								IF arrAxisCtrl[AxiseNo.AxisName.TailCurlLine].Cmd.arrbRealPoint[1] THEN
									IF Mach_Control.WJ_b.SinStepMode THEN//尾卷单步模式
									TailCurlSinStep:=TRUE;
								ELSE
									TailCurlSinStep:=FALSE;
								END_IF	
									arrAxisCtrl[AxiseNo.AxisName.TailCurlLine].Cmd.iGoSetPos:=0;
									//Mach_Control.WJ_b.TailCultOffloadingDone:=TRUE;
									TailCurlStep3:=1305;
								ELSE
									arrAxisCtrl[AxiseNo.AxisName.TailCurlLine].Cmd.iGoSetPos:=1;//尾卷夹电芯平移至初始位
								END_IF
						END_IF	
				END_IF	

				1305:
							IF NOT TailCurlSinStep THEN			
								IF 	arrAxisCtrl[AxiseNo.AxisName.TailCurlUpDown].Status.Homed AND arrAxisCtrl[AxiseNo.AxisName.TailCurlUpDown].Status.NoMoving  THEN
									IF arrAxisCtrl[AxiseNo.AxisName.TailCurlUpDown].Cmd.arrbRealPoint[4] THEN
													arrAxisCtrl[AxiseNo.AxisName.TailCurlUpDown].Cmd.iGoSetPos:=0;
													IF Mach_Control.WJ_b.SinStepMode THEN//尾卷单步模式
													TailCurlSinStep:=TRUE;
													ELSE
														TailCurlSinStep:=FALSE;
													END_IF	
													TailCurlStep3:=1310;
									ELSE
													arrAxisCtrl[AxiseNo.AxisName.TailCurlUpDown].Cmd.iGoSetPos:=4;//尾卷夹电芯升降至下电芯位
									END_IF
								END_IF	
						END_IF	
				
				1310:
					IF NOT TailCurlSinStep THEN		
					 IF arrAxisCtrl[AxiseNo.AxisName.GluingLine].Status.fActPos<=arrAxispar[AxiseNo.AxisName.GluingLine].arrTargetPoint[10] 
						AND arrAxisCtrl[AxiseNo.AxisName.GluingLine].Status.Homed AND NOT Mach_Control.WJ_b.TailCultOffloading AND arrAxis[AxiseNo.AxisName.TailCurlWhirling].Status.Homed 
						AND arrAxisCtrl[AxiseNo.AxisName.TailCurlWhirling].Status.NoMoving AND arrAxisCtrl[AxiseNo.AxisName.TailCurlLine].Status.NoMoving AND arrAxisCtrl[AxiseNo.AxisName.TailCurlLine].Cmd.arrbRealPoint[1] THEN
						
								IF arrAxisCtrl[AxiseNo.AxisName.TailCurlWhirling].Cmd.arrbRealPoint[1] THEN
									IF Mach_Control.WJ_b.SinStepMode THEN//尾卷单步模式
									TailCurlSinStep:=TRUE;
								ELSE
									TailCurlSinStep:=FALSE;
								END_IF	
									arrAxisCtrl[AxiseNo.AxisName.TailCurlWhirling].Cmd.iGoSetPos:=0;
									
									TailCurlStep3:=1320;
								ELSE
									arrAxisCtrl[AxiseNo.AxisName.TailCurlWhirling].Cmd.iGoSetPos:=1;//尾卷夹电芯旋转至取电芯位
								END_IF
						END_IF	
				END_IF	
	
	            1320://尾卷夹电芯平移去取电芯等待位
					 IF NOT TailCurlSinStep THEN	
								 IF  arrAxisCtrl[AxiseNo.AxisName.TailCurlUpDown].Status.Homed AND arrAxisCtrl[AxiseNo.AxisName.TailCurlUpDown].Status.NoMoving THEN
												IF arrAxisCtrl[AxiseNo.AxisName.TailCurlUpDown].Cmd.arrbRealPoint[1] THEN
													arrAxisCtrl[AxiseNo.AxisName.TailCurlUpDown].Cmd.iGoSetPos:=0;
												ELSE
													arrAxisCtrl[AxiseNo.AxisName.TailCurlUpDown].Cmd.iGoSetPos:=1;//尾卷夹升降去取电芯高度
												END_IF
								 END_IF
							 
							   IF arrAxisCtrl[AxiseNo.AxisName.TailCurlWhirling].Cmd.arrbRealPoint[1] AND arrAxisCtrl[AxiseNo.AxisName.TailCurlUpDown].Cmd.arrbRealPoint[1] AND
								  arrAxisCtrl[AxiseNo.AxisName.TailCurlSEPTALine].Cmd.arrbRealPoint[1] AND  arrAxisCtrl[AxiseNo.AxisName.TailCurlSEPTAUpDown].Cmd.arrbRealPoint[1] AND
								  arrAxisCtrl[AxiseNo.AxisName.LCurlingneedleLine].Cmd.arrbRealPoint[1] AND arrAxisCtrl[AxiseNo.AxisName.SCurlingneedleLine].Cmd.arrbRealPoint[1] AND
								  arrCyCtrl[arrCyNo.CylinderName.PoleSplintCy_D].Io.DIOFFSwitch AND arrCyCtrl[arrCyNo.CylinderName.TailCurlUpdownCy].Io.DIOFFSwitch AND
								  arrAxisCtrl[AxiseNo.AxisName.TailCurlLine].Status.Homed AND arrAxisCtrl[AxiseNo.AxisName.TailCurlLine].Status.NoMoving  THEN
									   IF arrAxisCtrl[AxiseNo.AxisName.TailCurlLine].Cmd.arrbRealPoint[11]  THEN
										  arrAxisCtrl[AxiseNo.AxisName.TailCurlLine].Cmd.iGoSetPos:=0;
											IF Mach_Control.WJ_b.SinStepMode THEN//尾卷单步模式
											   TailCurlSinStep:=TRUE;
											ELSE
											   TailCurlSinStep:=FALSE;
											END_IF									
											   TailCurlStep3:=0;
											   TailCurlTorMark:=FALSE;//尾卷夹电芯平移力矩判断标志位
									   ELSE
										   arrAxisCtrl[AxiseNo.AxisName.TailCurlLine].Cmd.iGoSetPos:=11;//尾卷夹电芯平移去取电芯等待位
										   TailCurlTorMark:=TRUE;//尾卷夹电芯平移力矩判断标志位
									   END_IF   
								END_IF
					  END_IF
	
	
	END_CASE	
ELSE
	//tailCult_GearInMultiMaster.Enable:=FALSE;//尾卷拉膜耦合放卷虚轴
//	tailCurlGearInEnable:=FALSE;//夹电芯平移轴与夹隔膜平移轴电子齿轮耦合
//	fbGearInGMvirbEnable	:=FALSE;	//隔膜纠䐔
;
END_IF	

CASE TailCurlStep3 OF 
	
		

	   200:
	   				IF NOT TailCurlSinStep THEN	
						
							hot_time_ton.IN:=TRUE;
							IF NOT arrCyCtrl[arrCyNo.CylinderName.PoleHotCutterCy].Cmd.bON AND NOT  arrCyCtrl[arrCyNo.CylinderName.PoleHotCutterCy].Status.ONState AND NOT hot_time_ton.Q THEN
								Mach_Control.WJ_b.HotCut:=TRUE;//启动热切
							END_IF
							
							IF hot_time_ton.Q THEN
							arrCyCtrl[arrCyNo.CylinderName.PoleHotCutterCy].Cmd.bON:=TRUE;//隔膜热切升降气缸伸出
							END_IF
							
							IF arrCyCtrl[arrCyNo.CylinderName.PoleHotCutterCy].Status.ONState  THEN
									Mach_Control.WJ_b.HotCut:=FALSE;//启动热切
									WJ_TON[1].IN:=FALSE;
									hot_time_ton.IN:=FALSE;
									TailCurlStep3:=205;	
								IF Mach_Control.WJ_b.SinStepMode THEN//尾卷单步模式
									TailCurlSinStep:=TRUE;
								ELSE
									TailCurlSinStep:=FALSE;
								END_IF								
							END_IF	
					END_IF
					


		305:
		
						
			SLCurlingneedleLine_TON.IN:=arrCyCtrl[arrCyNo.CylinderName.CurlingSplintCy_L].Status.OFFState AND arrCyCtrl[arrCyNo.CylinderName.CurlingSplintCy_S].Status.OFFState ;
				arrCyCtrl[arrCyNo.CylinderName.CurlingSplintCy_L].Cmd.bOFF:=TRUE;//尾卷长卷针张开
				arrCyCtrl[arrCyNo.CylinderName.CurlingSplintCy_S].Cmd.bOFF:=TRUE;//尾卷短卷针张开
				//arrCyCtrl[arrCyNo.CylinderName.CurlingSplintCy_S_1].Cmd.bON:=TRUE;//尾卷短卷针泄压关闭
				IF 	arrAxisCtrl[AxiseNo.AxisName.LCurlingneedleWhirling].Status.Homed AND arrAxisCtrl[AxiseNo.AxisName.LCurlingneedleWhirling].Status.NoMoving THEN
					IF arrAxisCtrl[AxiseNo.AxisName.LCurlingneedleWhirling].Cmd.arrbRealPoint[1] THEN
						arrAxisCtrl[AxiseNo.AxisName.LCurlingneedleWhirling].Cmd.iGoSetPos:=0;
					ELSE
						arrAxisCtrl[AxiseNo.AxisName.LCurlingneedleWhirling].Cmd.iGoSetPos:=1;//长卷针旋转至初始位
					END_IF
				END_IF										
				IF 	arrAxisCtrl[AxiseNo.AxisName.SCurlingneedleWhirling].Status.Homed AND arrAxisCtrl[AxiseNo.AxisName.SCurlingneedleWhirling].Status.NoMoving THEN
					IF arrAxisCtrl[AxiseNo.AxisName.SCurlingneedleWhirling].Cmd.arrbRealPoint[1] THEN
						arrAxisCtrl[AxiseNo.AxisName.SCurlingneedleWhirling].Cmd.iGoSetPos:=0;
					ELSE
						arrAxisCtrl[AxiseNo.AxisName.SCurlingneedleWhirling].Cmd.iGoSetPos:=1;//短卷针旋转至初始位
					END_IF
				END_IF
				IF 	 arrAxisCtrl[AxiseNo.AxisName.LCurlingneedleWhirling].Status.Moving AND arrAxisCtrl[AxiseNo.AxisName.SCurlingneedleWhirling].Status.Moving AND
					arrCyCtrl[arrCyNo.CylinderName.CurlingSplintCy_L].Status.OFFState AND arrCyCtrl[arrCyNo.CylinderName.CurlingSplintCy_S].Status.OFFState THEN														
					TailCurlStep3:=310;
				END_IF	
						

		1120:
	   				IF NOT TailCurlSinStep THEN	
						
							hot_time_ton.IN:=TRUE;
							IF NOT arrCyCtrl[arrCyNo.CylinderName.PoleHotCutterCy].Cmd.bON AND NOT  arrCyCtrl[arrCyNo.CylinderName.PoleHotCutterCy].Status.ONState AND NOT hot_time_ton.Q THEN
								Mach_Control.WJ_b.HotCut:=TRUE;//启动热切
							END_IF
							
							IF hot_time_ton.Q THEN
							arrCyCtrl[arrCyNo.CylinderName.PoleHotCutterCy].Cmd.bON:=TRUE;//隔膜热切升降气缸伸出
							END_IF
							
							IF arrCyCtrl[arrCyNo.CylinderName.PoleHotCutterCy].Status.ONState  THEN
									Mach_Control.WJ_b.HotCut:=FALSE;//启动热切
									WJ_TON[1].IN:=FALSE;
									hot_time_ton.IN:=FALSE;
									TailCurlStep3:=1140;	
								IF Mach_Control.WJ_b.SinStepMode THEN//尾卷单步模式
									TailCurlSinStep:=TRUE;
								ELSE
									TailCurlSinStep:=FALSE;
								END_IF								
							END_IF	
					END_IF			
				
				
				
END_CASE

 CASE TailCurlStep6 OF
10:
	IF (arrAxisCtrl[AxiseNo.AxisName.TailCurlSEPTALine].Status.fActPos<=(arrAxisPar[AxiseNo.AxisName.TailCurlSEPTALine].arrTargetPoint[1]+1)) OR Mach_Control.WJ_b.TailCurlDone  THEN
						 Mach_Control.DT_b.OffloadDone:=TRUE;
						 TailCurlStep6:=20;
					END_IF
					
20:
	TailCurlStep6:=666;

END_CASE 













//尾卷拉膜耦合放卷虚轴			
tailCult_GearInMultiMaster(
	Master1:=arrAxis[AxiseNo.AxisName.TailCurlRetracting] , 
	Master2:=arrAxis[AxiseNo.AxisName.TailCurlLine]  , 
	Master3:=arrAxis[AxiseNo.VirAxisName.VirDriver]  , 
	Master4:=arrAxis[AxiseNo.VirAxisName.VirDriver]  , 
	Slave:=arrAxis[AxiseNo.VirAxisName.VirDriver], 
	Enable:=tailCult_GearInMultiMaster.Enable , 
	GearRatio1:=-1 , 
	GearRatio2:=-1 , 
	GearRatio3:=0 , 
	GearRatio4:=0, 
	Acceleration:= , 
	Deceleration:= , 
	Jerk:= , 
	BufferMode:= , 
	Options:= , 
	InGear=> , 
	Busy=> , 
	Active=> , 
	CommandAborted=> , 
	Error=> , 
	ErrorID=> );				
tailCult_GearInMultiMaster.Error;
tailCult_GearInMultiMaster.Busy;	

//放卷虚轴解除耦合
fTailCurl_TRIG(CLK:=tailCult_GearInMultiMaster.Enable , Q=> );
tailCurl_CamOut(
	Slave:=arrAxis[AxiseNo.VirAxisName.VirDriver]  , 
	Execute:=fTailCurl_TRIG.Q , 
	Options:= , 
	Done=> , 
	Busy=> , 
	Error=> , 
	ErrorID=> );	
	
	
		
//夹电芯平移轴与夹隔膜平移轴电子齿轮耦合
	
	tailCurl_GearIn(
	Reset:=        stSysState.bReset  , 
	fratio1:= 1, 
	bError=> , 
	bReady=> , 
	InGear=> , 
	bEnable:=     tailCurlGearInEnable    , 
	master:=       arrAxis[AxiseNo.AxisName.TailCurlLine]  , 
	slave1:=        arrAxis[AxiseNo.AxisName.TailCurlSEPTALine], );
	tailCurl_GearIn.InGear;
	tailCurl_GearIn.bError;
	tailCurl_GearIn.bReady;
	
	
//夹电芯平移轴与夹隔膜平移轴电子齿轮耦合--取料
tailCurl_GearIn1.fratio1:=(arrAxisPar[AxiseNo.AxisName.TailCurlSEPTALine].arrTargetPoint[2]-arrAxisPar[AxiseNo.AxisName.TailCurlSEPTALine].arrTargetPoint[1])/(arrAxisPar[AxiseNo.AxisName.TailCurlLine].arrTargetPoint[2]-arrAxisPar[AxiseNo.AxisName.TailCurlLine].arrTargetPoint[11]);;
tailCurl_GearIn1(
	Reset:=        stSysState.bReset  , 
	fratio1:= , 
	bError=> , 
	bReady=> , 
	InGear=> , 
	bEnable:=     tailCurlGearInEnable1    , 
	master:=       arrAxis[AxiseNo.AxisName.TailCurlLine]  , 
	slave1:=        arrAxis[AxiseNo.AxisName.TailCurlSEPTALine], );
	tailCurl_GearIn1.InGear;
	tailCurl_GearIn1.bError;
	tailCurl_GearIn1.bReady;
		
	
	
//尾卷夹电芯伸缩取料齿轮耦合
tailRetGearIn.fratio1:=(arrAxisPar[AxiseNo.AxisName.TailCurlRetracting].arrTargetPoint[2]-arrAxisPar[AxiseNo.AxisName.TailCurlRetracting].arrTargetPoint[1])/(arrAxisPar[AxiseNo.AxisName.TailCurlLine].arrTargetPoint[2]-arrAxisPar[AxiseNo.AxisName.TailCurlLine].arrTargetPoint[11]);
	tailRetGearIn(
	Reset:=        stSysState.bReset  , 
	fratio1:= , 
	bError=> , 
	bReady=> , 
	InGear=> , 
	bEnable:=     tailRetGearInEnable    , 
	master:=       arrAxis[AxiseNo.AxisName.TailCurlLine]  , 
	slave1:=        arrAxis[AxiseNo.AxisName.TailCurlRetracting], );
	tailRetGearIn.InGear;
	tailRetGearIn.bError;
	tailRetGearIn.bReady;
	


//长、短卷针平移电子齿轮耦合  CurlingneedleLine    FB_GearInDyn
	CurlingneedleLine_GearIn(
	Reset:=        stSysState.bReset  , 
	fratio1:= -1, 
	bError=> , 
	bReady=> , 
	InGear=> , 
	bEnable:=     CurlingneedleLineEnable    , 
	master:=       arrAxis[AxiseNo.AxisName.LCurlingneedleLine]  , 
	slave1:=        arrAxis[AxiseNo.AxisName.SCurlingneedleLine], );
	
	CurlingneedleLine_GearIn.InGear;
	CurlingneedleLine_GearIn.bError;
	CurlingneedleLine_GearIn.bReady;
END_ACTION

ACTION TailCurl_Auto2:
//判断尾卷是否有轴在耕合中
IF arrAxisCtrl[AxiseNo.AxisName.TailCurlSEPTALine].Status.Coupled OR arrAxisCtrl[AxiseNo.AxisName.TailCurlSEPTAUpDown].Status.Coupled OR  
	arrAxisCtrl[AxiseNo.AxisName.LCurlingneedleWhirling].Status.Coupled OR arrAxisCtrl[AxiseNo.AxisName.SCurlingneedleWhirling].Status.Coupled THEN
	TailCurlCoupling:=TRUE;//尾卷轴耦合中
ELSE
	TailCurlCoupling:=FALSE;
END_IF



IF Mach_Control.U.WJ_iMode=1  THEN//在自动状态下
//尾卷电芯自动
		CASE TailCurlStep4 OF
			0://判断尾卷是否启动
					IF TailCurlStart THEN
						TailCurlStart:=FALSE;//复位尾卷启动
						Mach_Control.WJ_b.TailCurlDone:=FALSE;	//尾卷完成
						arrAxisCtrl[AxiseNo.VirAxisName.VirTailCurl].Cmd.bMoveAbs:=FALSE;//主轴启动
						TailCurlStep4:=10;
					END_IF
			10://尾卷凸轮耦合，判断尾卷主轴是停止、当前位置是否为0
				 	IF arrAxis[AxiseNo.VirAxisName.VirTailCurl].Status.NotMoving AND ABS(arrAxis[AxiseNo.VirAxisName.VirTailCurl].NcToPlc.ActPos)<=0.1 AND NOT TailCurlCoupling THEN
						TailCurlStep4:=30;
					ELSE
						TailCurlStep0:=50;
						TailCurlStep4:=20;			
					END_IF		
			20://等待主轴停止并且清零完成
					IF TailCurlStep0=6666 THEN
						TailCurlStep4:=30;	
					END_IF
					
			30://凸轮耦合
					fbCamInEndWindX.bCamInExecute:=TRUE;//夹膜平移轴凸轮耦合
					fbCamInEndWindY.bCamInExecute:=TRUE;//夹膜升降轴凸轮耦合
					tailCurl1_GearIn.Execute:=TRUE;//短卷针齿轮耦合
					tailCurl2_GearIn.Execute:=TRUE;//长卷针齿轮耦合
					IF arrAxisCtrl[AxiseNo.AxisName.TailCurlSEPTALine].Status.Coupled AND  arrAxisCtrl[AxiseNo.AxisName.TailCurlSEPTAUpDown].Status.Coupled AND   
						arrAxisCtrl[AxiseNo.AxisName.LCurlingneedleWhirling].Status.Coupled AND arrAxisCtrl[AxiseNo.AxisName.SCurlingneedleWhirling].Status.Coupled THEN
						TailCurlStep4:=40;	
					END_IF
			40://主轴启动
					arrAxisCtrl[AxiseNo.VirAxisName.VirTailCurl].Cmd.bDynamitcsParSel:=2;
					arrAxisCtrl[AxiseNo.VirAxisName.VirTailCurl].Cmd.fPositon_of_Abs:=359.5*Par.stWJ_date.SumNo;
					arrAxisPar[AxiseNo.VirAxisName.VirTailCurl].fTagatTime:=Par.stWJ_date.CoeSpeed;
					arrAxisCtrl[AxiseNo.VirAxisName.VirTailCurl].Cmd.bMoveAbs:=TRUE;
					TailCurlStep4:=50;	
					TailCurlStep5:=10;//夹膜平移超限凸轮解除耦合
			50://	解除夹隔平移、夹隔升降凸轮耦合	
				IF NOT TailCurlSinStep THEN
					IF arrAxisCtrl[AxiseNo.VirAxisName.VirTailCurl].Status.fSetPos=359.5*Par.stWJ_date.SumNo AND arrAxisCtrl[AxiseNo.VirAxisName.VirTailCurl].Status.NoMoving AND 
                       TailCurlStep5=6666 THEN				
						fbCamInEndWindX.bCamInExecute:=FALSE;//夹膜平移轴凸轮耦合					
						fbCamInEndWindY.bCamInExecute:=FALSE;//夹膜升降轴凸轮耦合
						IF NOT arrAxisCtrl[AxiseNo.AxisName.TailCurlSEPTALine].Status.Coupled AND NOT arrAxisCtrl[AxiseNo.AxisName.TailCurlSEPTAUpDown].Status.Coupled THEN
								IF Mach_Control.WJ_b.SinStepMode THEN//尾卷单步模式
									TailCurlSinStep:=TRUE;
								ELSE
									TailCurlSinStep:=FALSE;
								END_IF
							TailCurlStep0 :=50;
							TailCurlStep4:=60;	
						END_IF
					END_IF
				END_IF
			60:
				IF TailCurlStep0=6666 THEN
					Mach_Control.WJ_b.TailCurlDone	:=TRUE;	//尾卷完成
					TailCurlStep4:=0;
				END_IF
			(*60://压隔膜平移气缸伸出、压隔膜平移升降气缸	
				arrCyCtrl[arrCyNo.CylinderName.PoleSplintCy_D].Cmd.bOFF:=TRUE;//尾卷夹隔膜下夹板收回位
				//arrCyCtrl[arrCyNo.CylinderName.TailCurlLineCy].Cmd.bON:=TRUE;//尾卷压轮平移气缸伸出
				//IF arrCyCtrl[arrCyNo.CylinderName.TailCurlLineCy].Status.ONState THEN
					//arrCyCtrl[arrCyNo.CylinderName.TailCurlUpdownCy].Cmd.bON:=TRUE;//尾卷压轮升降气缸下降
					//IF arrCyCtrl[arrCyNo.CylinderName.TailCurlUpdownCy].Status.ONState THEN
						TailCurlStep4:=70;
				//	END_IF				
				//END_IF
			70://夹隔膜平移至初始位，夹隔膜升降至初始位
				
				IF arrCyCtrl[arrCyNo.CylinderName.PoleSplintCy_D].Status.OFFState THEN
						IF 	 arrAxisCtrl[AxiseNo.AxisName.TailCurlSEPTALine].Status.Homed AND arrAxisCtrl[AxiseNo.AxisName.TailCurlSEPTALine].Status.NoMoving THEN
							IF arrAxisCtrl[AxiseNo.AxisName.TailCurlSEPTALine].Cmd.arrbRealPoint[1] THEN
								arrAxisCtrl[AxiseNo.AxisName.TailCurlSEPTALine].Cmd.iGoSetPos:=0;
							ELSE
								arrAxisCtrl[AxiseNo.AxisName.TailCurlSEPTALine].Cmd.iGoSetPos:=1;//尾卷夹隔膜平移初始位
							END_IF
						END_IF	
						IF 	 arrAxisCtrl[AxiseNo.AxisName.TailCurlSEPTAUpDown].Status.Homed AND arrAxisCtrl[AxiseNo.AxisName.TailCurlSEPTAUpDown].Status.NoMoving THEN
							IF arrAxisCtrl[AxiseNo.AxisName.TailCurlSEPTAUpDown].Cmd.arrbRealPoint[1] THEN
								arrAxisCtrl[AxiseNo.AxisName.TailCurlSEPTAUpDown].Cmd.iGoSetPos:=0;
							ELSE
								arrAxisCtrl[AxiseNo.AxisName.TailCurlSEPTAUpDown].Cmd.iGoSetPos:=1;//尾卷夹隔膜升降初始位
							END_IF
						END_IF
						IF 	arrAxisCtrl[AxiseNo.AxisName.TailCurlSEPTALine].Cmd.arrbRealPoint[1] AND  arrAxisCtrl[AxiseNo.AxisName.TailCurlSEPTAUpDown].Cmd.arrbRealPoint[1]  THEN
							TailCurlStep0 :=50;
							Mach_Control.WJ_b.TailCurlDone	:=TRUE;	//尾卷完成
							TailCurlStep4:=0;
						END_IF	
				END_IF		
			80://启动主轴
					arrAxisCtrl[AxiseNo.VirAxisName.VirTailCurl].Cmd.bDynamitcsParSel:=2;
					arrAxisCtrl[AxiseNo.VirAxisName.VirTailCurl].Cmd.fPositon_of_Abs:=540;
					arrAxisPar[AxiseNo.VirAxisName.VirTailCurl].fTagatTime:=20;
					arrAxisCtrl[AxiseNo.VirAxisName.VirTailCurl].Cmd.bMoveAbs:=TRUE;	
					TailCurlStep4:=90;
			90://判断主轴运动是否完成
					IF arrAxisCtrl[AxiseNo.VirAxisName.VirTailCurl].Status.fSetPos=540 AND arrAxisCtrl[AxiseNo.VirAxisName.VirTailCurl].Status.NoMoving THEN
							tailCurl1_GearIn.Execute:=FALSE;//短卷针齿轮耦合
							tailCurl2_GearIn.Execute:=FALSE;//长卷针齿轮耦合
							IF NOT arrAxisCtrl[AxiseNo.AxisName.LCurlingneedleWhirling].Status.Coupled AND NOT arrAxisCtrl[AxiseNo.AxisName.SCurlingneedleWhirling].Status.Coupled  THEN
								Mach_Control.WJ_b.TailCurlDone	:=TRUE;	//尾卷完成
								TailCurlStep0 :=50;
								TailCurlStep4:=0;	
							END_IF
					END_IF	*)		
		END_CASE
		
//尾卷主轴停止，当前位置清零
		CASE TailCurlStep0 OF
				50:
					TailCurlStep0:=100;
					
				100://判断主轴是否在运动中
					IF NOT TailCurlSinStep THEN
						IF arrAxis[AxiseNo.VirAxisName.VirTailCurl].Status.NotMoving  THEN
							arrAxisCtrl[AxiseNo.VirAxisName.VirTailCurl].Cmd.bStop:=FALSE;
							TailCurlStep0:=110;
								IF Mach_Control.WJ_b.SinStepMode THEN//尾卷单步模式
												TailCurlSinStep:=TRUE;
											ELSE
												TailCurlSinStep:=FALSE;
											END_IF
						ELSE
							arrAxisCtrl[AxiseNo.VirAxisName.VirTailCurl].Cmd.bStop:=TRUE;//尾卷主轴停止
						END_IF
						END_IF
				110://判断尾卷轴是否在耦合中
					IF NOT TailCurlSinStep THEN
						IF TailCurlCoupling  THEN
								TailCurlStep0:=120;
										IF Mach_Control.WJ_b.SinStepMode THEN//尾卷单步模式
												TailCurlSinStep:=TRUE;
											ELSE
												TailCurlSinStep:=FALSE;
											END_IF
						ELSE
								TailCurlStep0:=130;
										IF Mach_Control.WJ_b.SinStepMode THEN//尾卷单步模式
												TailCurlSinStep:=TRUE;
											ELSE
												TailCurlSinStep:=FALSE;
											END_IF
						END_IF
						END_IF
				120://尾卷凸轮解除耦合
						fbCamInEndWindX.bCamInExecute:=FALSE;
						fbCamInEndWindY.bCamInExecute:=FALSE;
						tailCurl1_GearIn.Execute:=FALSE;//短卷针齿轮耦合
						tailCurl2_GearIn.Execute:=FALSE;//长卷针齿轮耦合
						IF  NOT TailCurlCoupling THEN
							TailCurlStep0:=125;
						END_IF
						
				125:
					IF NOT TailCurlSinStep THEN
						arrAxisCtrl[AxiseNo.AxisName.TailCurlSEPTALine].Cmd.bStop:=TRUE;
						IF arrAxisCtrl[AxiseNo.AxisName.TailCurlSEPTALine].Status.NoMoving AND NOT arrAxisCtrl[AxiseNo.AxisName.TailCurlSEPTALine].Status.Coupled THEN
							
							IF Mach_Control.WJ_b.SinStepMode THEN//尾卷单步模式
								TailCurlSinStep:=TRUE;
							ELSE
								TailCurlSinStep:=FALSE;
							END_IF	
							arrAxisCtrl[AxiseNo.AxisName.TailCurlSEPTALine].Cmd.bStop:=FALSE;
							TailCurlStep0:=130;
						END_IF
					END_IF
				130://主轴当前位置清零
						IF NOT arrAxisCtrl[AxiseNo.AxisName.TailCurlSEPTALine].Status.Coupled AND 
							NOT arrAxisCtrl[AxiseNo.AxisName.TailCurlSEPTAUpDown].Status.Coupled THEN
									arrAxisCtrl[AxiseNo.VirAxisName.VirTailCurl].Cmd.fSetPos:=0;
									arrAxisCtrl[AxiseNo.VirAxisName.VirTailCurl].Cmd.bSetPos:=TRUE;	
									TailCurlStep0:=140;
						END_IF
				140://判断主轴清零是否完成
						//IF arrAxis[AxiseNo.VirAxisName.VirTailCurl].Status.NotMoving  AND arrAxis[AxiseNo.VirAxisName.VirTailCurl].NcToPlc.SetPos=0 THEN		
							TailCurlStep0:=150;
						//END_IF
						
						
				150:
					arrAxisCtrl[AxiseNo.VirAxisName.VirTailCurl].Cmd.bEnable:=FALSE;
					WJ_TON[3](IN:=NOT arrAxisCtrl[AxiseNo.VirAxisName.VirTailCurl].Cmd.bEnable, PT:=T#20MS, Q=> , ET=> );	
					IF WJ_TON[3].Q  THEN
						arrAxisCtrl[AxiseNo.VirAxisName.VirTailCurl].Cmd.bSetPos:=FALSE;
						arrAxisCtrl[AxiseNo.VirAxisName.VirTailCurl].Cmd.bStop:=FALSE;	
						WJ_TON[3](IN:=FALSE);	
						TailCurlStep0:=160;
					END_IF
				160:
					WJ_TON[4](IN:=FALSE);	
					arrAxisCtrl[AxiseNo.VirAxisName.VirTailCurl].Cmd.bEnable:=TRUE;	
					TailCurlStep0:=170;
				170:
					arrAxisCtrl[AxiseNo.VirAxisName.VirTailCurl].Cmd.bReset:=TRUE;
					WJ_TON[4](IN:=TRUE, PT:=T#20MS, Q=> , ET=> );	
					IF WJ_TON[4].Q THEN
						WJ_TON[4](IN:=FALSE);	
						TailCurlStep0:=180;
					END_IF
				180:	
					arrAxisCtrl[AxiseNo.VirAxisName.VirTailCurl].Cmd.bReset:=FALSE;	
					TailCurlStep0:=190;
						
				190:		
					IF arrAxis[AxiseNo.VirAxisName.VirTailCurl].Status.NotMoving  AND arrAxis[AxiseNo.VirAxisName.VirTailCurl].NcToPlc.SetPos=0 
						AND arrAxisCtrl[AxiseNo.VirAxisName.VirTailCurl].Cmd.bEnable THEN
						TailCurlStep0:=6666;
					END_IF		
						
		END_CASE
END_IF


CASE  TailCurlStep5 OF
10:
	IF arrAxisCtrl[AxiseNo.VirAxisName.VirTailCurl].Status.fActPos>0  AND arrAxisCtrl[AxiseNo.AxisName.TailCurlSEPTALine].Status.fSetPos<=(par.stWJ_date.WJ_PoistCamOut+2 ) 
		AND arrAxisCtrl[AxiseNo.VirAxisName.VirTailCurl].Status.fActPos<=357 THEN//解耦
		fbCamInEndWindX.bGearOutMode:=TRUE;//夹膜平移轴凸轮耦合
		fbCamInEndWindX.bCamInExecute:=FALSE;//夹膜平移轴凸轮耦合
		
		IF NOT fbCamInEndWindX.bCamInExecute THEN
			TailCurlStep5:=100;
		END_IF
	ELSIF arrAxisCtrl[AxiseNo.VirAxisName.VirTailCurl].Status.fActPos>357 AND arrAxisCtrl[AxiseNo.AxisName.TailCurlSEPTALine].Status.fSetPos>=par.stWJ_date.WJ_PoistCamOut THEN//不解耦
		TailCurlStep5:=6666;
	END_IF
	
100:
	IF NOT  fbCamInEndWindX.bCamInExecute AND NOT arrAxisCtrl[AxiseNo.AxisName.TailCurlSEPTALine].Status.Coupled AND NOT fbCamInEndWindX.bInSync  THEN
		TailCurlStep5:=200;
	END_IF
200://高速定位停止
	arrAxisCtrl[AxiseNo.AxisName.TailCurlSEPTALine].Cmd.bDynamitcsParSel:=2;
	arrAxisCtrl[AxiseNo.AxisName.TailCurlSEPTALine].Cmd.fPositon_of_Abs:=par.stWJ_date.WJ_PoistCamOut-1;
	arrAxisPar[AxiseNo.AxisName.TailCurlSEPTALine].fTagatTime:= 0.02;//3.33333/arrAxisPar[AxiseNo.AxisName.TailCurlSEPTALine].fVelocity_of_Abs+0.01 
	arrAxisCtrl[AxiseNo.AxisName.TailCurlSEPTALine].Cmd.bMoveAbs:=TRUE;
	TailCurlStep5:=300;
300:
	IF ABS(arrAxisCtrl[AxiseNo.AxisName.TailCurlSEPTALine].Status.fActPos+1-par.stWJ_date.WJ_PoistCamOut)<=0.5 AND NOT arrAxisCtrl[AxiseNo.AxisName.TailCurlSEPTALine].Cmd.bMoveAbs
	AND arrAxisCtrl[AxiseNo.AxisName.TailCurlSEPTALine].Status.NoMoving THEN
		arrAxisCtrl[AxiseNo.AxisName.TailCurlSEPTALine].Cmd.bMoveAbs:=FALSE;
		TailCurlStep5:=400;
	END_IF
400:
	arrAxisCtrl[AxiseNo.AxisName.TailCurlSEPTALine].Cmd.bDynamitcsParSel:=1;
	fbCamInEndWindX.bGearOutMode:=FALSE;//夹膜平移轴凸轮耦合
	IF arrAxisCtrl[AxiseNo.AxisName.TailCurlSEPTALine].Cmd.bDynamitcsParSel=1 THEN
		TailCurlStep5:=6666;
	END_IF
END_CASE

(*
CASE  TailCurlStep5 OF
			10:
					IF 	 arrAxisCtrl[AxiseNo.VirAxisName.VirTailCurl].Status.fActPos>0  AND arrAxisCtrl[AxiseNo.AxisName.TailCurlSEPTALine].Status.fSetPos<=par.stWJ_date.WJ_PoistCamOut   THEN
							fbCamInEndWindX.bCamInExecute:=FALSE;//夹膜平移轴凸轮耦合
							//arrAxisCtrl[AxiseNo.AxisName.SEPTATLine].Cmd.bStop:=TRUE;
					END_IF
					IF NOT fbCamInEndWindX.bCamInExecute THEN
						TailCurlStep5:=6666;
					END_IF
END_CASE
*)
(**************************************夹膜平移正常解耦位计算******************************************************)
arrAxisPar[AxiseNo.AxisName.TailCurlSEPTALine].arrTargetPoint[4]:=arrAxisPar[AxiseNo.AxisName.TailCurlSEPTALine].arrTargetPoint[2]
								-(arrAxisPar[AxiseNo.AxisName.TailCurlLine].arrTargetPoint[7]-arrAxisPar[AxiseNo.AxisName.TailCurlLine].arrTargetPoint[4])
								-(fbRoll_New.AxisXmm*2);
END_ACTION

ACTION TailCurl_Condition:
//尾卷夹电芯平移轴移动至初始位置的安全件件
(*
IF  arrAxis[AxiseNo.AxisName.TailCurlWhirling].Status.Homed AND arrAxisCtrl[AxiseNo.AxisName.TailCurlWhirling].Status.NoMoving AND
	(arrAxisCtrl[AxiseNo.AxisName.TailCurlWhirling].Cmd.arrbRealPoint[1] OR arrAxisCtrl[AxiseNo.AxisName.TailCurlWhirling].Cmd.arrbRealPoint[2]) AND	
	arrAxisCtrl[AxiseNo.AxisName.LCurlingneedleLine].Status.Homed AND arrAxisCtrl[AxiseNo.AxisName.LCurlingneedleLine].Status.NoMoving AND arrAxisCtrl[AxiseNo.AxisName.LCurlingneedleLine].Cmd.arrbRealPoint[1] AND 
	arrAxisCtrl[AxiseNo.AxisName.SCurlingneedleLine].Status.Homed AND arrAxisCtrl[AxiseNo.AxisName.SCurlingneedleLine].Status.NoMoving AND arrAxisCtrl[AxiseNo.AxisName.SCurlingneedleLine].Cmd.arrbRealPoint[1]  
OR Mach_Control.WJ_b.AxisConditionEN THEN
	arrAxisCtrl[AxiseNo.AxisName.TailCurlLine].Cmd.GoPoint_Condition[1]:=TRUE;
ELSE
	arrAxisCtrl[AxiseNo.AxisName.TailCurlLine].Cmd.GoPoint_Condition[1]:=FALSE;
END_IF

//尾卷夹隔膜轴移动至取电芯位的安全条件
IF arrAxisCtrl[AxiseNo.AxisName.CaDTCarryingLine].Status.Homed AND arrAxisCtrl[AxiseNo.AxisName.CaDTCarryingLine].Status.NoMoving AND arrAxisCtrl[AxiseNo.AxisName.CaDTCarryingLine].Cmd.arrbRealPoint[1] 
OR Mach_Control.WJ_b.AxisConditionEN THEN	
	arrAxisCtrl[AxiseNo.AxisName.TailCurlSEPTALine].Cmd.GoPoint_Condition[2]:=TRUE;
ELSE
	arrAxisCtrl[AxiseNo.AxisName.TailCurlSEPTALine].Cmd.GoPoint_Condition[2]:=FALSE;	
END_IF
*)

/////////////////////////////////////////////////////////////
/////////////////////////////////////////////////////////
////////////////////////////////////////////电机条件
//尾卷夹电芯平移 
IF  Mach_Control.U.WJ_iMode=3 AND 
	arrAxisCtrl[AxiseNo.AxisName.LCurlingneedleLine].Status.fActPos<=arrAxisPar[AxiseNo.AxisName.LCurlingneedleLine].arrTargetPoint[1]+1 AND arrAxisCtrl[AxiseNo.AxisName.LCurlingneedleLine].Status.Homed  AND
	arrAxisCtrl[AxiseNo.AxisName.SCurlingneedleLine].Status.fActPos <=arrAxisPar[AxiseNo.AxisName.SCurlingneedleLine] .arrTargetPoint[1]+1 AND arrAxisCtrl[AxiseNo.AxisName.SCurlingneedleLine].Status.Homed AND 
	(arrAxisCtrl[AxiseNo.AxisName.TailCurlWhirling].Status.fActPos<=arrAxisPar[AxiseNo.AxisName.TailCurlWhirling].arrTargetPoint[1]+1 AND
	arrAxisCtrl[AxiseNo.AxisName.TailCurlWhirling].Status.fActPos>=arrAxisPar[AxiseNo.AxisName.TailCurlWhirling].arrTargetPoint[1]-1	) OR 
	(arrAxisCtrl[AxiseNo.AxisName.TailCurlWhirling].Status.fActPos<=arrAxisPar[AxiseNo.AxisName.TailCurlWhirling].arrTargetPoint[2]+1 AND
	arrAxisCtrl[AxiseNo.AxisName.TailCurlWhirling].Status.fActPos>=arrAxisPar[AxiseNo.AxisName.TailCurlWhirling].arrTargetPoint[2]-1	) 
    OR Mach_Control.WJ_b.AxisConditionEN THEN
	arrAxisCtrl[AxiseNo.AxisName.TailCurlLine].Cmd.Home_Condition:=TRUE;
ELSE
	arrAxisCtrl[AxiseNo.AxisName.TailCurlLine].Cmd.Home_Condition:=FALSE;	
END_IF

IF Mach_Control.U.WJ_iMode=3 AND
	arrAxisCtrl[AxiseNo.AxisName.LCurlingneedleLine].Status.fActPos<=arrAxisPar[AxiseNo.AxisName.LCurlingneedleLine].arrTargetPoint[1]+1 AND arrAxisCtrl[AxiseNo.AxisName.LCurlingneedleLine].Status.Homed  AND
	arrAxisCtrl[AxiseNo.AxisName.SCurlingneedleLine].Status.fActPos <=arrAxisPar[AxiseNo.AxisName.SCurlingneedleLine] .arrTargetPoint[1]+1 AND arrAxisCtrl[AxiseNo.AxisName.SCurlingneedleLine].Status.Homed 
 THEN
   arrAxisCtrl[AxiseNo.AxisName.TailCurlLine].Cmd.JogP_Condition:=TRUE;
   arrAxisCtrl[AxiseNo.AxisName.TailCurlLine].Cmd.JogN_Condition:=TRUE;
   ELSE 
   arrAxisCtrl[AxiseNo.AxisName.TailCurlLine].Cmd.JogP_Condition:=FALSE;
   arrAxisCtrl[AxiseNo.AxisName.TailCurlLine].Cmd.JogN_Condition:=FALSE;
 END_IF

IF  Mach_Control.U.WJ_iMode=3 AND arrAxisCtrl[AxiseNo.AxisName.TailCurlLine].Status.Homed 
AND (arrAxisCtrl[AxiseNo.AxisName.TailCurlWhirling].Cmd.arrbRealPoint[1] OR  arrAxisCtrl[AxiseNo.AxisName.TailCurlWhirling].Cmd.arrbRealPoint[2]) AND
arrAxisCtrl[AxiseNo.AxisName.LCurlingneedleLine].Status.fActPos<=arrAxisPar[AxiseNo.AxisName.LCurlingneedleLine].arrTargetPoint[1]+1 AND arrAxisCtrl[AxiseNo.AxisName.LCurlingneedleLine].Status.Homed  AND
arrAxisCtrl[AxiseNo.AxisName.SCurlingneedleLine].Status.fActPos <=arrAxisPar[AxiseNo.AxisName.SCurlingneedleLine] .arrTargetPoint[1]+1 AND arrAxisCtrl[AxiseNo.AxisName.SCurlingneedleLine].Status.Homed 
OR Mach_Control.WJ_b.AxisConditionEN THEN
	arrAxisCtrl[AxiseNo.AxisName.TailCurlLine].Cmd.GoPoint_Condition[1]:=TRUE;
ELSE
	arrAxisCtrl[AxiseNo.AxisName.TailCurlLine].Cmd.GoPoint_Condition[1]:=FALSE;	
END_IF

IF  Mach_Control.U.WJ_iMode=3 AND arrAxisCtrl[AxiseNo.AxisName.TailCurlLine].Status.Homed 
AND (arrAxisCtrl[AxiseNo.AxisName.TailCurlWhirling].Cmd.arrbRealPoint[1]
AND NOT arrAxisCtrl[AxiseNo.AxisName.TailCurlWhirling].Cmd.arrbRealPoint[2]
AND arrAxisCtrl[AxiseNo.AxisName.TailCurlSEPTAUpDown].Cmd.arrbRealPoint[1]  
AND  arrCyCtrl[arrCyNo.CylinderName.PoleHotCutterCy].Status.OFFState
AND  arrAxisCtrl[AxiseNo.AxisName.LCurlingneedleLine].Status.fActPos<=arrAxisPar[AxiseNo.AxisName.LCurlingneedleLine].arrTargetPoint[1]+1 AND arrAxisCtrl[AxiseNo.AxisName.LCurlingneedleLine].Status.Homed  
AND arrAxisCtrl[AxiseNo.AxisName.SCurlingneedleLine].Status.fActPos <=arrAxisPar[AxiseNo.AxisName.SCurlingneedleLine] .arrTargetPoint[1]+1 AND arrAxisCtrl[AxiseNo.AxisName.SCurlingneedleLine].Status.Homed 
AND arrAxisCtrl[AxiseNo.AxisName.TailCurlUpDown].Cmd.arrbRealPoint[1] )
AND  arrCyCtrl[arrCyNo.CylinderName.TailCurlSplintCy].Io.DIOFFSwitch 
AND arrCyCtrl[arrCyNo.CylinderName.PoleSplintCy_D].Status.OFFState
AND arrAxisCtrl[AxiseNo.AxisName.TailCurlSEPTALine].Cmd.arrbRealPoint[2]
AND  arrAxisCtrl[AxiseNo.AxisName.SEPTATLine].Cmd.arrbRealPoint[1] 
  OR Mach_Control.WJ_b.AxisConditionEN THEN
	arrAxisCtrl[AxiseNo.AxisName.TailCurlLine].Cmd.GoPoint_Condition[2]:=TRUE;
ELSE
	arrAxisCtrl[AxiseNo.AxisName.TailCurlLine].Cmd.GoPoint_Condition[2]:=FALSE;	
END_IF

IF  Mach_Control.U.WJ_iMode=3 AND arrAxisCtrl[AxiseNo.AxisName.TailCurlLine].Status.Homed 
AND (arrAxisCtrl[AxiseNo.AxisName.TailCurlWhirling].Cmd.arrbRealPoint[1] 
AND NOT  arrAxisCtrl[AxiseNo.AxisName.TailCurlWhirling].Cmd.arrbRealPoint[2]) 
AND  arrAxisCtrl[AxiseNo.AxisName.LCurlingneedleLine].Status.fActPos<=arrAxisPar[AxiseNo.AxisName.LCurlingneedleLine].arrTargetPoint[1]+1 AND arrAxisCtrl[AxiseNo.AxisName.LCurlingneedleLine].Status.Homed  
AND  arrAxisCtrl[AxiseNo.AxisName.SCurlingneedleLine].Status.fActPos <=arrAxisPar[AxiseNo.AxisName.SCurlingneedleLine] .arrTargetPoint[1]+1 AND arrAxisCtrl[AxiseNo.AxisName.SCurlingneedleLine].Status.Homed 
OR Mach_Control.WJ_b.AxisConditionEN THEN
	arrAxisCtrl[AxiseNo.AxisName.TailCurlLine].Cmd.GoPoint_Condition[3]:=TRUE;
ELSE
	arrAxisCtrl[AxiseNo.AxisName.TailCurlLine].Cmd.GoPoint_Condition[3]:=FALSE;	
END_IF

IF  Mach_Control.U.WJ_iMode=3 AND arrAxisCtrl[AxiseNo.AxisName.TailCurlLine].Status.Homed 
AND arrAxisCtrl[AxiseNo.AxisName.TailCurlWhirling].Cmd.arrbRealPoint[1] 
AND arrAxisCtrl[AxiseNo.AxisName.LCurlingneedleLine].Status.fActPos<=arrAxisPar[AxiseNo.AxisName.LCurlingneedleLine].arrTargetPoint[1] +1
AND arrAxisCtrl[AxiseNo.AxisName.LCurlingneedleLine].Status.Homed  
AND arrAxisCtrl[AxiseNo.AxisName.SCurlingneedleLine].Status.fActPos <=arrAxisPar[AxiseNo.AxisName.SCurlingneedleLine] .arrTargetPoint[1]+1 
AND arrAxisCtrl[AxiseNo.AxisName.SCurlingneedleLine].Status.Homed 
OR Mach_Control.WJ_b.AxisConditionEN THEN
	arrAxisCtrl[AxiseNo.AxisName.TailCurlLine].Cmd.GoPoint_Condition[4]:=TRUE;
ELSE
	arrAxisCtrl[AxiseNo.AxisName.TailCurlLine].Cmd.GoPoint_Condition[4]:=FALSE;	
END_IF

IF  Mach_Control.U.WJ_iMode=3 AND arrAxisCtrl[AxiseNo.AxisName.TailCurlLine].Status.Homed  
AND arrAxisCtrl[AxiseNo.AxisName.TailCurlWhirling].Cmd.arrbRealPoint[1] 
AND arrAxisCtrl[AxiseNo.AxisName.LCurlingneedleLine].Status.fActPos<=arrAxisPar[AxiseNo.AxisName.LCurlingneedleLine].arrTargetPoint[1]+1 
AND arrAxisCtrl[AxiseNo.AxisName.LCurlingneedleLine].Status.Homed  
AND arrAxisCtrl[AxiseNo.AxisName.SCurlingneedleLine].Status.fActPos <=arrAxisPar[AxiseNo.AxisName.SCurlingneedleLine] .arrTargetPoint[1]+1 
AND arrAxisCtrl[AxiseNo.AxisName.SCurlingneedleLine].Status.Homed 
OR Mach_Control.WJ_b.AxisConditionEN THEN
	arrAxisCtrl[AxiseNo.AxisName.TailCurlLine].Cmd.GoPoint_Condition[5]:=TRUE;
ELSE
	arrAxisCtrl[AxiseNo.AxisName.TailCurlLine].Cmd.GoPoint_Condition[5]:=FALSE;	
END_IF

IF  Mach_Control.U.WJ_iMode=3 AND arrAxisCtrl[AxiseNo.AxisName.TailCurlLine].Status.Homed 
AND arrAxisCtrl[AxiseNo.AxisName.TailCurlWhirling].Cmd.arrbRealPoint[2] 
AND arrAxisCtrl[AxiseNo.AxisName.LCurlingneedleLine].Status.fActPos<=arrAxisPar[AxiseNo.AxisName.LCurlingneedleLine].arrTargetPoint[1]+1 
AND arrAxisCtrl[AxiseNo.AxisName.LCurlingneedleLine].Status.Homed  
AND arrAxisCtrl[AxiseNo.AxisName.SCurlingneedleLine].Status.fActPos <=arrAxisPar[AxiseNo.AxisName.SCurlingneedleLine] .arrTargetPoint[1]+1 
AND arrAxisCtrl[AxiseNo.AxisName.SCurlingneedleLine].Status.Homed 
AND arrCyCtrl[arrCyNo.CylinderName.PullGlueModelCy].Status.ONState
OR Mach_Control.WJ_b.AxisConditionEN THEN
	arrAxisCtrl[AxiseNo.AxisName.TailCurlLine].Cmd.GoPoint_Condition[6]:=TRUE;
ELSE
	arrAxisCtrl[AxiseNo.AxisName.TailCurlLine].Cmd.GoPoint_Condition[6]:=FALSE;	
END_IF

IF  Mach_Control.U.WJ_iMode=3 AND arrAxisCtrl[AxiseNo.AxisName.TailCurlLine].Status.Homed 
AND arrAxisCtrl[AxiseNo.AxisName.TailCurlWhirling].Cmd.arrbRealPoint[1] 
AND arrAxisCtrl[AxiseNo.AxisName.TailCurlSEPTAUpDown].Cmd.arrbRealPoint[1]  
AND arrAxisCtrl[AxiseNo.AxisName.LCurlingneedleLine].Status.fActPos<=arrAxisPar[AxiseNo.AxisName.LCurlingneedleLine].arrTargetPoint[1] +1
AND arrAxisCtrl[AxiseNo.AxisName.LCurlingneedleLine].Status.Homed  
AND arrAxisCtrl[AxiseNo.AxisName.SCurlingneedleLine].Status.fActPos <=arrAxisPar[AxiseNo.AxisName.SCurlingneedleLine] .arrTargetPoint[1]+1 
AND arrAxisCtrl[AxiseNo.AxisName.SCurlingneedleLine].Status.Homed 
AND arrAxisCtrl[AxiseNo.AxisName.TailCurlSEPTALine].Cmd.arrbRealPoint[2]
OR Mach_Control.WJ_b.AxisConditionEN THEN
	arrAxisCtrl[AxiseNo.AxisName.TailCurlLine].Cmd.GoPoint_Condition[7]:=TRUE;
ELSE
	arrAxisCtrl[AxiseNo.AxisName.TailCurlLine].Cmd.GoPoint_Condition[7]:=FALSE;	
END_IF

IF  Mach_Control.U.WJ_iMode=3 AND arrAxisCtrl[AxiseNo.AxisName.TailCurlLine].Status.Homed  
AND arrAxisCtrl[AxiseNo.AxisName.TailCurlWhirling].Cmd.arrbRealPoint[1] 
AND arrAxisCtrl[AxiseNo.AxisName.LCurlingneedleLine].Status.fActPos<=arrAxisPar[AxiseNo.AxisName.LCurlingneedleLine].arrTargetPoint[1]+1 
AND arrAxisCtrl[AxiseNo.AxisName.LCurlingneedleLine].Status.Homed  
AND arrAxisCtrl[AxiseNo.AxisName.SCurlingneedleLine].Status.fActPos <=arrAxisPar[AxiseNo.AxisName.SCurlingneedleLine] .arrTargetPoint[1]+1 
AND arrAxisCtrl[AxiseNo.AxisName.SCurlingneedleLine].Status.Homed  THEN
	arrAxisCtrl[AxiseNo.AxisName.TailCurlLine].Cmd.GoPoint_Condition[8]:=TRUE;
ELSE
	arrAxisCtrl[AxiseNo.AxisName.TailCurlLine].Cmd.GoPoint_Condition[8]:=FALSE;	
END_IF

IF  Mach_Control.U.WJ_iMode=3 AND   arrAxisCtrl[AxiseNo.AxisName.TailCurlLine].Status.Homed  
AND  arrAxisCtrl[AxiseNo.AxisName.TailCurlWhirling].Cmd.arrbRealPoint[1] 
AND(arrAxisCtrl[AxiseNo.AxisName.LCurlingneedleLine].Status.fActPos<=arrAxisPar[AxiseNo.AxisName.LCurlingneedleLine].arrTargetPoint[1]+1 
AND arrAxisCtrl[AxiseNo.AxisName.LCurlingneedleLine].Status.Homed  
AND arrAxisCtrl[AxiseNo.AxisName.SCurlingneedleLine].Status.fActPos <=arrAxisPar[AxiseNo.AxisName.SCurlingneedleLine] .arrTargetPoint[1]+1 
AND arrAxisCtrl[AxiseNo.AxisName.SCurlingneedleLine].Status.Homed 
AND arrCyCtrl[arrCyNo.CylinderName.PoleSplintCy_D].Status.OFFState
AND arrAxisCtrl[AxiseNo.AxisName.TailCurlSEPTALine].Cmd.arrbRealPoint[2]
AND arrAxisCtrl[AxiseNo.AxisName.TailCurlSEPTAUpDown].Cmd.arrbRealPoint[1] ) OR Mach_Control.WJ_b.AxisConditionEN THEN
    arrAxisCtrl[AxiseNo.AxisName.TailCurlLine].Cmd.GoPoint_Condition[9]:=TRUE;
ELSE
	arrAxisCtrl[AxiseNo.AxisName.TailCurlLine].Cmd.GoPoint_Condition[9]:=FALSE;	
END_IF

IF  Mach_Control.U.WJ_iMode=3 AND arrAxisCtrl[AxiseNo.AxisName.TailCurlLine].Status.Homed 
AND arrAxisCtrl[AxiseNo.AxisName.TailCurlWhirling].Cmd.arrbRealPoint[1] 
AND arrAxisCtrl[AxiseNo.AxisName.LCurlingneedleLine].Status.fActPos<=arrAxisPar[AxiseNo.AxisName.LCurlingneedleLine].arrTargetPoint[1] +1
AND arrAxisCtrl[AxiseNo.AxisName.LCurlingneedleLine].Status.Homed  
AND arrAxisCtrl[AxiseNo.AxisName.SCurlingneedleLine].Status.fActPos <=arrAxisPar[AxiseNo.AxisName.SCurlingneedleLine] .arrTargetPoint[1] +1
AND arrAxisCtrl[AxiseNo.AxisName.SCurlingneedleLine].Status.Homed 
OR Mach_Control.WJ_b.AxisConditionEN THEN
	arrAxisCtrl[AxiseNo.AxisName.TailCurlLine].Cmd.GoPoint_Condition[10]:=TRUE;
ELSE
	arrAxisCtrl[AxiseNo.AxisName.TailCurlLine].Cmd.GoPoint_Condition[10]:=FALSE;	
END_IF

IF  Mach_Control.U.WJ_iMode=3 AND   arrAxisCtrl[AxiseNo.AxisName.TailCurlLine].Status.Homed  AND   arrAxisCtrl[AxiseNo.AxisName.TailCurlWhirling].Cmd.arrbRealPoint[1] AND
	(arrAxisCtrl[AxiseNo.AxisName.LCurlingneedleLine].Status.fActPos<=arrAxisPar[AxiseNo.AxisName.LCurlingneedleLine].arrTargetPoint[1]+1 AND arrAxisCtrl[AxiseNo.AxisName.LCurlingneedleLine].Status.Homed  AND
	arrAxisCtrl[AxiseNo.AxisName.SCurlingneedleLine].Status.fActPos <=arrAxisPar[AxiseNo.AxisName.SCurlingneedleLine] .arrTargetPoint[1]+1 AND arrAxisCtrl[AxiseNo.AxisName.SCurlingneedleLine].Status.Homed  AND
	arrAxisCtrl[AxiseNo.AxisName.TailCurlSEPTAUpDown].Cmd.arrbRealPoint[1] ) AND  arrCyCtrl[arrCyNo.CylinderName.PoleSplintCy_D].Status.OFFState AND
    arrAxisCtrl[AxiseNo.AxisName.TailCurlSEPTALine].Cmd.arrbRealPoint[1] OR Mach_Control.WJ_b.AxisConditionEN THEN
    arrAxisCtrl[AxiseNo.AxisName.TailCurlLine].Cmd.GoPoint_Condition[11]:=TRUE;
ELSE
	arrAxisCtrl[AxiseNo.AxisName.TailCurlLine].Cmd.GoPoint_Condition[11]:=FALSE;	
END_IF


//尾卷夹电芯伸缩
IF  Mach_Control.U.WJ_iMode=3  
OR Mach_Control.WJ_b.AxisConditionEN THEN
	arrAxisCtrl[AxiseNo.AxisName.TailCurlRetracting].Cmd.Home_Condition:=TRUE;
ELSE
	arrAxisCtrl[AxiseNo.AxisName.TailCurlRetracting].Cmd.Home_Condition:=FALSE;	
END_IF

IF  Mach_Control.U.WJ_iMode=3 AND arrAxisCtrl[AxiseNo.AxisName.TailCurlRetracting].Status.Homed 
OR Mach_Control.WJ_b.AxisConditionEN THEN
	arrAxisCtrl[AxiseNo.AxisName.TailCurlRetracting].Cmd.GoPoint_Condition[1]:=TRUE;
ELSE
	arrAxisCtrl[AxiseNo.AxisName.TailCurlRetracting].Cmd.GoPoint_Condition[1]:=FALSE;	
END_IF

IF  Mach_Control.U.WJ_iMode=3 AND arrAxisCtrl[AxiseNo.AxisName.TailCurlRetracting].Status.Homed 
OR Mach_Control.WJ_b.AxisConditionEN THEN
	arrAxisCtrl[AxiseNo.AxisName.TailCurlRetracting].Cmd.GoPoint_Condition[2]:=TRUE;
ELSE
	arrAxisCtrl[AxiseNo.AxisName.TailCurlRetracting].Cmd.GoPoint_Condition[2]:=FALSE;	
END_IF

IF  Mach_Control.U.WJ_iMode=3 AND arrAxisCtrl[AxiseNo.AxisName.TailCurlRetracting].Status.Homed 
OR Mach_Control.WJ_b.AxisConditionEN THEN
	arrAxisCtrl[AxiseNo.AxisName.TailCurlRetracting].Cmd.GoPoint_Condition[3]:=TRUE;
ELSE
	arrAxisCtrl[AxiseNo.AxisName.TailCurlRetracting].Cmd.GoPoint_Condition[3]:=FALSE;	
END_IF


//尾卷夹膜平移
IF  Mach_Control.U.WJ_iMode=3 AND
    arrAxisCtrl[AxiseNo.AxisName.CaDTCarryingUpDown].Status.fActPos<=arrAxisPar[AxiseNo.AxisName.CaDTCarryingUpDown].arrTargetPoint[5]+1 AND arrAxisCtrl[AxiseNo.AxisName.CaDTCarryingUpDown].Status.Homed AND
	arrAxisCtrl[AxiseNo.AxisName.CaDTCarryingLine].Status.Homed AND arrAxisCtrl[AxiseNo.AxisName.CaDTCarryingLine].Cmd.arrbRealPoint[1] 	 THEN
       arrAxisCtrl[AxiseNo.AxisName.TailCurlSEPTALine].Cmd.JogP_Condition:=TRUE;
ELSE 
	   arrAxisCtrl[AxiseNo.AxisName.TailCurlSEPTALine].Cmd.JogP_Condition:=FALSE;
END_IF 
 
IF  Mach_Control.U.WJ_iMode=3 AND
	arrAxisCtrl[AxiseNo.AxisName.TailCurlLine].Status.fActPos<=arrAxisPar[AxiseNo.AxisName.TailCurlLine].arrTargetPoint[4]+1 AND arrAxisCtrl[AxiseNo.AxisName.TailCurlLine].Status.Homed 
    OR Mach_Control.WJ_b.AxisConditionEN THEN
		arrAxisCtrl[AxiseNo.AxisName.TailCurlSEPTALine].Cmd.Home_Condition:=TRUE;
		arrAxisCtrl[AxiseNo.AxisName.TailCurlSEPTALine].Cmd.GoPoint_Condition[1]:=TRUE;
		//TailCurlSEPTALineGoargee:=TRUE;
ELSE
		arrAxisCtrl[AxiseNo.AxisName.TailCurlSEPTALine].Cmd.Home_Condition:=FALSE;	
		arrAxisCtrl[AxiseNo.AxisName.TailCurlSEPTALine].Cmd.GoPoint_Condition[1]:=FALSE;
		//TailCurlSEPTALineGoargee:=FALSE;
END_IF

IF  Mach_Control.U.WJ_iMode=3 AND
	arrAxisCtrl[AxiseNo.AxisName.CaDTCarryingUpDown].Status.fActPos<=arrAxisPar[AxiseNo.AxisName.CaDTCarryingUpDown].arrTargetPoint[5]+1 AND arrAxisCtrl[AxiseNo.AxisName.CaDTCarryingUpDown].Status.Homed AND
	arrAxisCtrl[AxiseNo.AxisName.CaDTCarryingLine].Status.Homed AND arrAxisCtrl[AxiseNo.AxisName.CaDTCarryingLine].Cmd.arrbRealPoint[1] 
OR Mach_Control.WJ_b.AxisConditionEN THEN
		arrAxisCtrl[AxiseNo.AxisName.TailCurlSEPTALine].Cmd.Home_Condition:=TRUE;

		arrAxisCtrl[AxiseNo.AxisName.TailCurlSEPTALine].Cmd.GoPoint_Condition[2]:=TRUE;
		//TailCurlSEPTALineGoargee:=TRUE;
ELSE
		arrAxisCtrl[AxiseNo.AxisName.TailCurlSEPTALine].Cmd.Home_Condition:=FALSE;	

		arrAxisCtrl[AxiseNo.AxisName.TailCurlSEPTALine].Cmd.GoPoint_Condition[2]:=FALSE;
		//TailCurlSEPTALineGoargee:=FALSE;
END_IF

(*
IF  Mach_Control.U.DT_iMode=3 AND arrAxisCtrl[AxiseNo.AxisName.CaCarryingLine2].Cmd.arrbRealPoint[1] 
AND (arrAxisCtrl[AxiseNo.AxisName.TailCurlLine].Cmd.arrbRealPoint[5] OR arrAxisCtrl[AxiseNo.AxisName.TailCurlLine].Cmd.arrbRealPoint[6] OR arrAxisCtrl[AxiseNo.AxisName.TailCurlLine].Cmd.arrbRealPoint[1])
AND (arrAxisCtrl[AxiseNo.AxisName.TailCurlWhirling].Cmd.arrbRealPoint[1] OR  arrAxisCtrl[AxiseNo.AxisName.TailCurlWhirling].Cmd.arrbRealPoint[2]) THEN
	arrAxisCtrl[AxiseNo.AxisName.TailCurlSEPTALine].Cmd.GoPoint_Condition[1]:=TRUE;
ELSE
	arrAxisCtrl[AxiseNo.AxisName.TailCurlSEPTALine].Cmd.GoPoint_Condition[1]:=FALSE;	
END_IF

IF  Mach_Control.U.DT_iMode=3 AND arrAxisCtrl[AxiseNo.AxisName.CaCarryingLine2].Cmd.arrbRealPoint[1] 
AND (arrAxisCtrl[AxiseNo.AxisName.TailCurlLine].Cmd.arrbRealPoint[5] OR arrAxisCtrl[AxiseNo.AxisName.TailCurlLine].Cmd.arrbRealPoint[6] OR arrAxisCtrl[AxiseNo.AxisName.TailCurlLine].Cmd.arrbRealPoint[1])
AND (arrAxisCtrl[AxiseNo.AxisName.TailCurlWhirling].Cmd.arrbRealPoint[1] OR  arrAxisCtrl[AxiseNo.AxisName.TailCurlWhirling].Cmd.arrbRealPoint[2]) THEN
	arrAxisCtrl[AxiseNo.AxisName.TailCurlSEPTALine].Cmd.GoPoint_Condition[2]:=TRUE;
ELSE
	arrAxisCtrl[AxiseNo.AxisName.TailCurlSEPTALine].Cmd.GoPoint_Condition[2]:=FALSE;	
END_IF
*)

//尾卷夹膜升降
IF  Mach_Control.U.WJ_iMode=3 AND
	 arrAxisCtrl[AxiseNo.AxisName.TailCurlLine].Status.fSetPos<=arrAxisPar[AxiseNo.AxisName.TailCurlLine].arrTargetPoint[4] AND arrAxisCtrl[AxiseNo.AxisName.TailCurlLine].Status.Homed    
OR Mach_Control.WJ_b.AxisConditionEN THEN
		arrAxisCtrl[AxiseNo.AxisName.TailCurlSEPTAUpDown].Cmd.Home_Condition:=TRUE;
ELSE
	arrAxisCtrl[AxiseNo.AxisName.TailCurlSEPTAUpDown].Cmd.Home_Condition:=FALSE;	
END_IF

IF  Mach_Control.U.WJ_iMode=3 AND arrAxisCtrl[AxiseNo.AxisName.TailCurlSEPTAUpDown].Status.Homed 
AND NOT arrAxisCtrl[AxiseNo.AxisName.TailCurlLine].Cmd.arrbRealPoint[11] OR Mach_Control.WJ_b.AxisConditionEN THEN
	arrAxisCtrl[AxiseNo.AxisName.TailCurlSEPTAUpDown].Cmd.GoPoint_Condition[1]:=TRUE;
ELSE
	arrAxisCtrl[AxiseNo.AxisName.TailCurlSEPTAUpDown].Cmd.GoPoint_Condition[1]:=FALSE;	
END_IF

IF  Mach_Control.U.WJ_iMode=3 AND arrAxisCtrl[AxiseNo.AxisName.TailCurlSEPTAUpDown].Status.Homed  
AND arrAxisCtrl[AxiseNo.AxisName.TailCurlLine].Status.fActPos <=  arrAxisPar[AxiseNo.AxisName.TailCurlLine].arrTargetPoint[4]  
AND NOT arrAxisCtrl[AxiseNo.AxisName.TailCurlLine].Cmd.arrbRealPoint[11] OR Mach_Control.WJ_b.AxisConditionEN THEN
	arrAxisCtrl[AxiseNo.AxisName.TailCurlSEPTAUpDown].Cmd.GoPoint_Condition[2]:=TRUE;
ELSE
	arrAxisCtrl[AxiseNo.AxisName.TailCurlSEPTAUpDown].Cmd.GoPoint_Condition[2]:=FALSE;	
END_IF

//尾卷夹电芯升降
IF  Mach_Control.U.WJ_iMode=3 AND  arrAxisCtrl[AxiseNo.AxisName.TailCurlRetracting].Cmd.arrbRealPoint[1] 
OR Mach_Control.WJ_b.AxisConditionEN THEN
	arrAxisCtrl[AxiseNo.AxisName.TailCurlUpDown].Cmd.Home_Condition:=TRUE;
ELSE
	arrAxisCtrl[AxiseNo.AxisName.TailCurlUpDown].Cmd.Home_Condition:=FALSE;	
END_IF

IF  Mach_Control.U.WJ_iMode=3 
AND arrAxisCtrl[AxiseNo.AxisName.TailCurlSEPTAUpDown].Status.Homed  
AND  arrAxisCtrl[AxiseNo.AxisName.TailCurlRetracting].Cmd.arrbRealPoint[1] 
AND NOT arrAxisCtrl[AxiseNo.AxisName.TailCurlLine].Cmd.arrbRealPoint[6]
OR Mach_Control.WJ_b.AxisConditionEN THEN
	arrAxisCtrl[AxiseNo.AxisName.TailCurlUpDown].Cmd.GoPoint_Condition[1]:=TRUE;
ELSE
	arrAxisCtrl[AxiseNo.AxisName.TailCurlUpDown].Cmd.GoPoint_Condition[1]:=FALSE;	
END_IF
////////////////////////////////////////////
IF  Mach_Control.U.WJ_iMode=3 
AND arrAxisCtrl[AxiseNo.AxisName.TailCurlSEPTAUpDown].Status.Homed  
AND arrAxisCtrl[AxiseNo.AxisName.TailCurlWhirling].Cmd.arrbRealPoint[1]
AND arrAxisCtrl[AxiseNo.AxisName.TailCurlRetracting].Cmd.arrbRealPoint[1] 
AND  arrAxisCtrl[AxiseNo.AxisName.TailCurlLine].Status.fActPos <=  arrAxisPar[AxiseNo.AxisName.TailCurlLine].arrTargetPoint[4]  
OR Mach_Control.WJ_b.AxisConditionEN THEN
	arrAxisCtrl[AxiseNo.AxisName.TailCurlUpDown].Cmd.GoPoint_Condition[2]:=TRUE;
ELSE
	arrAxisCtrl[AxiseNo.AxisName.TailCurlUpDown].Cmd.GoPoint_Condition[2]:=FALSE;	
END_IF

IF  Mach_Control.U.WJ_iMode=3 
AND arrAxisCtrl[AxiseNo.AxisName.TailCurlSEPTAUpDown].Status.Homed 
AND arrAxisCtrl[AxiseNo.AxisName.TailCurlRetracting].Cmd.arrbRealPoint[1]
AND NOT arrAxisCtrl[AxiseNo.AxisName.TailCurlLine].Cmd.arrbRealPoint[11] 
OR Mach_Control.WJ_b.AxisConditionEN THEN
	arrAxisCtrl[AxiseNo.AxisName.TailCurlUpDown].Cmd.GoPoint_Condition[3]:=TRUE;

ELSE
	arrAxisCtrl[AxiseNo.AxisName.TailCurlUpDown].Cmd.GoPoint_Condition[3]:=FALSE;	
END_IF

IF  Mach_Control.U.WJ_iMode=3 
AND arrAxisCtrl[AxiseNo.AxisName.TailCurlSEPTAUpDown].Status.Homed
AND arrAxisCtrl[AxiseNo.AxisName.TailCurlWhirling].Cmd.arrbRealPoint[2]  
AND arrAxisCtrl[AxiseNo.AxisName.TailCurlRetracting].Cmd.arrbRealPoint[1]
AND NOT arrAxisCtrl[AxiseNo.AxisName.TailCurlLine].Cmd.arrbRealPoint[11] 
OR Mach_Control.WJ_b.AxisConditionEN THEN
	arrAxisCtrl[AxiseNo.AxisName.TailCurlUpDown].Cmd.GoPoint_Condition[4]:=TRUE;
ELSE
	arrAxisCtrl[AxiseNo.AxisName.TailCurlUpDown].Cmd.GoPoint_Condition[4]:=FALSE;	
END_IF
///////////////////////////////////////////
//尾卷夹电芯旋转 
IF  Mach_Control.U.WJ_iMode=3 AND  arrAxisCtrl[AxiseNo.AxisName.TailCurlRetracting].Cmd.arrbRealPoint[1] AND arrAxisCtrl[AxiseNo.AxisName.TailCurlLine].Cmd.arrbRealPoint[1] AND
   arrAxisCtrl[AxiseNo.AxisName.TailCurlRetracting].Status.Homed AND arrAxisCtrl[AxiseNo.AxisName.TailCurlLine].Status.Homed 	
OR Mach_Control.WJ_b.AxisConditionEN THEN
	arrAxisCtrl[AxiseNo.AxisName.TailCurlWhirling].Cmd.Home_Condition:=TRUE;
ELSE
	arrAxisCtrl[AxiseNo.AxisName.TailCurlWhirling].Cmd.Home_Condition:=FALSE;	
END_IF

IF  Mach_Control.U.WJ_iMode=3 AND arrAxis[AxiseNo.AxisName.TailCurlWhirling].Status.Homed  AND  arrAxisCtrl[AxiseNo.AxisName.TailCurlRetracting].Cmd.arrbRealPoint[1] 
AND arrAxisCtrl[AxiseNo.AxisName.TailCurlUpDown].Cmd.arrbRealPoint[3] AND arrAxisCtrl[AxiseNo.AxisName.TailCurlLine].Cmd.arrbRealPoint[1] 
OR Mach_Control.WJ_b.AxisConditionEN THEN
	arrAxisCtrl[AxiseNo.AxisName.TailCurlWhirling].Cmd.GoPoint_Condition[1]:=TRUE;
ELSE
	arrAxisCtrl[AxiseNo.AxisName.TailCurlWhirling].Cmd.GoPoint_Condition[1]:=FALSE;	
END_IF

IF  Mach_Control.U.WJ_iMode=3 AND arrAxis[AxiseNo.AxisName.TailCurlWhirling].Status.Homed  AND  arrAxisCtrl[AxiseNo.AxisName.TailCurlRetracting].Cmd.arrbRealPoint[1] 
AND arrAxisCtrl[AxiseNo.AxisName.TailCurlUpDown].Cmd.arrbRealPoint[3] AND arrAxisCtrl[AxiseNo.AxisName.TailCurlLine].Cmd.arrbRealPoint[1] 
OR Mach_Control.WJ_b.AxisConditionEN THEN
	arrAxisCtrl[AxiseNo.AxisName.TailCurlWhirling].Cmd.GoPoint_Condition[2]:=TRUE;
ELSE
	arrAxisCtrl[AxiseNo.AxisName.TailCurlWhirling].Cmd.GoPoint_Condition[2]:=FALSE;	
END_IF

//尾卷长卷针平移
IF  Mach_Control.U.WJ_iMode=3 
OR Mach_Control.WJ_b.AxisConditionEN THEN
	arrAxisCtrl[AxiseNo.AxisName.LCurlingneedleLine].Cmd.Home_Condition:=TRUE;
ELSE
	arrAxisCtrl[AxiseNo.AxisName.LCurlingneedleLine].Cmd.Home_Condition:=FALSE;	
END_IF

IF  Mach_Control.U.WJ_iMode=3 AND arrAxisCtrl[AxiseNo.AxisName.LCurlingneedleLine].Status.Homed AND arrCyCtrl[arrCyNo.CylinderName.CurlingSplintCy_L].Status.OFFState
OR Mach_Control.WJ_b.AxisConditionEN THEN
	arrAxisCtrl[AxiseNo.AxisName.LCurlingneedleLine].Cmd.GoPoint_Condition[1]:=TRUE;
ELSE
	arrAxisCtrl[AxiseNo.AxisName.LCurlingneedleLine].Cmd.GoPoint_Condition[1]:=FALSE;	
END_IF

IF  Mach_Control.U.WJ_iMode=3 AND arrAxisCtrl[AxiseNo.AxisName.LCurlingneedleLine].Status.Homed AND arrCyCtrl[arrCyNo.CylinderName.CurlingSplintCy_L].Status.OFFState
     AND  arrAxisCtrl[AxiseNo.AxisName.TailCurlLine].Cmd.arrbRealPoint[4]   OR Mach_Control.WJ_b.AxisConditionEN THEN
	arrAxisCtrl[AxiseNo.AxisName.LCurlingneedleLine].Cmd.GoPoint_Condition[2]:=TRUE;
ELSE
	arrAxisCtrl[AxiseNo.AxisName.LCurlingneedleLine].Cmd.GoPoint_Condition[2]:=FALSE;	
END_IF


//尾卷短卷针平移
IF  (Mach_Control.U.WJ_iMode=3  AND arrAxisCtrl[AxiseNo.AxisName.SCurlingneedleWhirling].Io.biHomeSwitch)
OR Mach_Control.WJ_b.AxisConditionEN   THEN
	arrAxisCtrl[AxiseNo.AxisName.SCurlingneedleLine].Cmd.Home_Condition:=TRUE;
ELSE
	arrAxisCtrl[AxiseNo.AxisName.SCurlingneedleLine].Cmd.Home_Condition:=FALSE;	
END_IF

IF  Mach_Control.U.WJ_iMode=3 AND arrAxisCtrl[AxiseNo.AxisName.SCurlingneedleLine].Status.Homed  AND arrCyCtrl[arrCyNo.CylinderName.CurlingSplintCy_S].Status.OFFState
OR Mach_Control.WJ_b.AxisConditionEN THEN
	arrAxisCtrl[AxiseNo.AxisName.SCurlingneedleLine].Cmd.GoPoint_Condition[1]:=TRUE;
ELSE
	arrAxisCtrl[AxiseNo.AxisName.SCurlingneedleLine].Cmd.GoPoint_Condition[1]:=FALSE;	
END_IF

IF  Mach_Control.U.WJ_iMode=3 AND arrAxisCtrl[AxiseNo.AxisName.SCurlingneedleLine].Status.Homed  AND arrCyCtrl[arrCyNo.CylinderName.CurlingSplintCy_S].Status.OFFState
    AND  arrCyCtrl[arrCyNo.ElectValveName.WJShortvacuum].Io.DOStatus1 AND  arrAxisCtrl[AxiseNo.AxisName.TailCurlLine].Cmd.arrbRealPoint[4]    OR Mach_Control.WJ_b.AxisConditionEN THEN
	arrAxisCtrl[AxiseNo.AxisName.SCurlingneedleLine].Cmd.GoPoint_Condition[2]:=TRUE;
ELSE
	arrAxisCtrl[AxiseNo.AxisName.SCurlingneedleLine].Cmd.GoPoint_Condition[2]:=FALSE;	
END_IF

//尾卷长卷针旋转
IF  Mach_Control.U.WJ_iMode=3 AND arrAxisCtrl[AxiseNo.AxisName.LCurlingneedleLine].Status.fSetPos<=arrAxisPar[AxiseNo.AxisName.LCurlingneedleLine].arrTargetPoint[1]  
OR Mach_Control.WJ_b.AxisConditionEN THEN
	arrAxisCtrl[AxiseNo.AxisName.LCurlingneedleWhirling].Cmd.Home_Condition:=TRUE;
ELSE
	arrAxisCtrl[AxiseNo.AxisName.LCurlingneedleWhirling].Cmd.Home_Condition:=FALSE;	
END_IF

IF  Mach_Control.U.WJ_iMode=3 AND arrAxisCtrl[AxiseNo.AxisName.LCurlingneedleWhirling].Status.Homed 
AND arrAxisCtrl[AxiseNo.AxisName.LCurlingneedleLine].Cmd.arrbRealPoint[1]  
OR Mach_Control.WJ_b.AxisConditionEN THEN
	arrAxisCtrl[AxiseNo.AxisName.LCurlingneedleWhirling].Cmd.GoPoint_Condition[1]:=TRUE;
ELSE
	arrAxisCtrl[AxiseNo.AxisName.LCurlingneedleWhirling].Cmd.GoPoint_Condition[1]:=FALSE;	
END_IF

//尾卷短卷针旋转
IF  Mach_Control.U.WJ_iMode=3 AND arrAxisCtrl[AxiseNo.AxisName.SCurlingneedleLine].Status.fSetPos<=arrAxisPar[AxiseNo.AxisName.SCurlingneedleLine].arrTargetPoint[1]  
OR Mach_Control.WJ_b.AxisConditionEN THEN
	arrAxisCtrl[AxiseNo.AxisName.SCurlingneedleWhirling].Cmd.Home_Condition:=TRUE;
ELSE
	arrAxisCtrl[AxiseNo.AxisName.SCurlingneedleWhirling].Cmd.Home_Condition:=FALSE;	
END_IF

IF  Mach_Control.U.WJ_iMode=3 AND arrAxisCtrl[AxiseNo.AxisName.SCurlingneedleWhirling].Status.Homed 
AND arrAxisCtrl[AxiseNo.AxisName.SCurlingneedleLine].Cmd.arrbRealPoint[1]  
OR Mach_Control.WJ_b.AxisConditionEN THEN
	arrAxisCtrl[AxiseNo.AxisName.SCurlingneedleWhirling].Cmd.GoPoint_Condition[1]:=TRUE;
ELSE
	arrAxisCtrl[AxiseNo.AxisName.SCurlingneedleWhirling].Cmd.GoPoint_Condition[1]:=FALSE;	
END_IF
END_ACTION

ACTION TailCurl_Gohome:
Tailcurl_GohomeOverTon(IN:= , PT:=T#90S , Q=> , ET=> );//叠台回原点超时报警延时

//判断回原点的状态
IF arrAxisCtrl[AxiseNo.AxisName.SCurlingneedleLine].Status.Homed AND arrAxisCtrl[AxiseNo.AxisName.LCurlingneedleLine].Status.Homed AND 
	arrAxisCtrl[AxiseNo.AxisName.LCurlingneedleWhirling].Status.Homed  AND arrAxisCtrl[AxiseNo.AxisName.SCurlingneedleWhirling].Status.Homed AND 
	arrAxisCtrl[AxiseNo.AxisName.TailCurlLine].Status.Homed AND arrAxisCtrl[AxiseNo.AxisName.TailCurlRetracting].Status.Homed AND 
	arrAxisCtrl[AxiseNo.AxisName.TailCurlUpDown].Status.Homed AND arrAxisCtrl[AxiseNo.AxisName.TailCurlSEPTAUpDown].Status.Homed AND 
	arrAxis[AxiseNo.AxisName.TailCurlSEPTALine].Status.Homed AND arrAxis[AxiseNo.AxisName.TailCurlWhirling].Status.Homed AND WZIniti_Done THEN
		Mach_Control.WJ_b.WZIniti_Done:=TRUE;//初始化完成	
ELSE
		Mach_Control.WJ_b.WZIniti_Done:=FALSE;//初始化完成	
END_IF

IF Mach_Control.U.WJ_iMode=3 THEN//在手动状态下
	IF  Tailcurl_Gohoming THEN
			IF 	NOT Tailcurl_GohomeOverTon.Q THEN
				    Tailcurl_GohomeOverTon.IN:=TRUE;
			ELSE
				IF 	Tailcurl_GohomeOverTon.Q THEN
					Tailcurl_Gohoming:=FALSE;
					TailCurlStep1:=0;
				     Mach_Control.WJ_b.Error[19]:=TRUE;//尾卷回原点超时报警
				     Tailcurl_GohomeOverTon.IN:=FALSE;
				END_IF	 
					 
			END_IF
	
	ELSE
			Tailcurl_GohomeOverTon.IN:=FALSE;
	END_IF
	
	IF r_TailCurl_init.Q THEN
		Tailcurl_GohomeDone:=FALSE;//尾卷回原点完成
		Tailcurl_Gohoming:=FALSE;//尾卷回原点中
		TailCurlStep1:=0;
		Mach_Control.WJ_b.WZIniti_Done:=FALSE;//负极取片回原点完成
		WZIniti_Done:=FALSE;//负极取片回原点完成
	END_IF	

	//尾卷贴胶初始化
	r_TailCurl_init(CLK:=Mach_Control.WJ_b.WZIniti_Hbtn , Q=> );
	f_TailCurl_init(CLK:=Mach_Control.WJ_b.WZIniti_Hbtn   , Q=> );
	tTailCurlTON(IN:= , PT:=T#0.5S , Q=> , ET=> );
	CASE TailCurlStep1 OF
	0://启动尾卷贴胶初始化，气缸复位
		IF f_TailCurl_init.Q THEN	
			Tailcurl_GohomeDone:=FALSE;//尾卷回原点完成
		    Tailcurl_Gohoming:=TRUE;//尾卷回原点中
			TailCurlStep1:=1;
		END_IF
	1://回原点完成复位
			WZIniti_Done:=FALSE;//初始化完成	
			TailCurlStep3 :=0;
			TailCurlStep4:=0;
			TailCurlStep5:=0;
			TailCurlStep6:=0;
			
			arrAxisCtrl[AxiseNo.AxisName.TailCurlSEPTALine].Cmd.fOverride:=100;
			arrAxisCtrl[AxiseNo.AxisName.TailCurlRetracting].Cmd.fOverride:=100;
			arrAxisCtrl[AxiseNo.AxisName.TailCurlLine].Cmd.fOverride:=100;
						
			tailCult_GearInMultiMaster.Enable:=FALSE;
			tailCurlGearInEnable:=FALSE;
			tailCurlGearInEnable1:=FALSE;
			tailRetGearInEnable:=FALSE;//夹电芯平移与夹电芯伸缩电子齿轮
			CurlingneedleLineEnable:=FALSE;
			tailCult_GearInMultiMaster.Enable:=FALSE;
			
			 Mach_Control.DT_b.OffloadDone:=FALSE;
			 Mach_Control.WJ_b.TailCurlDone	:=FALSE;
			 //Mach_Control.DT_b.OffloadRequest:=FALSE;//复位电芯下料请求	
			 Mach_Control.WJ_b.TailCultOffloading:=FALSE;
			CellMemory[Mach_Control.WJ_b.WJ_Memory].Cell:=FALSE;	
			TailCurlStart:=FALSE;//复位尾卷启动
			Mach_Control.WJ_b.TailCurlDone	:=FALSE;	//尾卷完成
			arrAxisCtrl[AxiseNo.VirAxisName.VirTailCurl].Cmd.bMoveAbs:=FALSE;//主轴启动
			CurlingneedleLineEnable:=FALSE;//长、短卷针平移电子齿轮耦合启动
			tailCurlGearInEnable:=FALSE;//电子齿轮耦合		
			tTailCurlTON.IN:=FALSE;
			arrAxisCtrl[AxiseNo.AxisName.TailCurlSEPTALine].Cmd.bDynamitcsParSel:=1;
			fbCamInEndWindX.bGearOutMode:=FALSE;//夹膜平移轴凸轮耦合
			IF NOT WZIniti_Done AND arrAxisCtrl[AxiseNo.AxisName.TailCurlSEPTALine].Cmd.bDynamitcsParSel=1 THEN
				TailCurlStep1:=10;
			END_IF
	10://气缸复位，尾卷状态复位
			IF  NOT 	tTailCurlTON.Q THEN	
					tTailCurlTON.IN:=TRUE;
					//arrCyCtrl[arrCyNo.CylinderName.CurlingSplintCy_S_1].Cmd.bON:=TRUE;//尾卷短卷针泄压关闭
					arrCyCtrl[arrCyNo.CylinderName.CurlingSplintCy_L].Cmd.bOFF:=TRUE;//尾卷长卷针张开
					arrCyCtrl[arrCyNo.CylinderName.CurlingSplintCy_S].Cmd.bOFF:=TRUE;//尾卷短卷针张开	
					arrCyCtrl[arrCyNo.ElectValveName.WJShortvacuum].Cmd.bON:=TRUE;//短卷针张开真空开
					arrCyCtrl[arrCyNo.CylinderName.PoleHotCutterCy].Cmd.bOFF:=TRUE;//隔膜热切升降气缸收回
					arrCyCtrl[arrCyNo.CylinderName.PoleSplintCy_D].Cmd.bOFF:=TRUE;//隔膜隔膜下夹板气缸收回
					arrCyCtrl[arrCyNo.CylinderName.TailCurlUpdownCy].Cmd.bOFF:=TRUE;//尾卷压轮升降气缸收回
					arrCyCtrl[arrCyNo.CylinderName.TailCurlSplintCy].Cmd.bOFF:=TRUE;//尾卷取料夹爪气缸张开	
			ELSE
					IF arrCyCtrl[arrCyNo.CylinderName.PoleHotCutterCy].Io.DIOFFSwitch AND arrCyCtrl[arrCyNo.CylinderName.PoleSplintCy_D].Io.DIOFFSwitch AND 
					   arrCyCtrl[arrCyNo.CylinderName.TailCurlUpdownCy].Io.DIOFFSwitch AND arrCyCtrl[arrCyNo.CylinderName.TailCurlSplintCy].Io.DIOFFSwitch THEN
					   tTailCurlTON.IN:=FALSE;
					   TailCurlStep1:=20;
					END_IF	
			END_IF	
	20:
			fbCamInEndWindX.bCamInExecute:=FALSE;//夹膜平移凸轮耦合
			fbCamInEndWindY.bCamInExecute:=FALSE;//夹膜升降凸轮耦合
			tailCurl1_GearIn.Execute:=FALSE;//短卷针齿轮耦合
			tailCurl2_GearIn.Execute:=FALSE;//长卷针齿轮耦合
			IF NOT fbCamInEndWindX.bCamInExecute AND NOT fbCamInEndWindY.bCamInExecute AND 
				NOT tailCurl1_GearIn.Execute AND NOT tailCurl2_GearIn.Execute THEN
				TailCurlStep1:=21;
			END_IF
	21://解除凸轮耦合
			arrCyCtrl[arrCyNo.CylinderName.TailCurlLineCy].Cmd.bOFF:=TRUE;//尾卷压轮平移气缸收回
			arrAxisCtrl[AxiseNo.AxisName.SCurlingneedleWhirling].Cmd.bGearOut:=TRUE;//尾卷短卷针旋转轴解耦
			arrAxisCtrl[AxiseNo.AxisName.LCurlingneedleWhirling].Cmd.bGearOut:=TRUE;//尾卷长卷针旋转轴解耦
			arrAxisCtrl[AxiseNo.AxisName.TailCurlLine].Cmd.bGearOut:=TRUE;//尾卷夹电芯平移轴解耦
			arrAxisCtrl[AxiseNo.AxisName.TailCurlSEPTALine].Cmd.bGearOut:=TRUE;//尾卷夹膜平移轴解耦 
			arrAxisCtrl[AxiseNo.AxisName.TailCurlSEPTAUpDown].Cmd.bGearOut:=TRUE;//尾卷夹膜升降轴解耦 
			IF NOT arrAxisCtrl[AxiseNo.AxisName.SCurlingneedleWhirling].Status.Coupled AND  NOT arrAxisCtrl[AxiseNo.AxisName.LCurlingneedleWhirling].Status.Coupled AND 
				NOT arrAxisCtrl[AxiseNo.AxisName.TailCurlLine].Status.Coupled AND NOT arrAxisCtrl[AxiseNo.AxisName.TailCurlSEPTALine].Status.Coupled AND 
				NOT arrAxisCtrl[AxiseNo.AxisName.TailCurlSEPTAUpDown].Status.Coupled THEN
				TailCurlStep1:=25;
			END_IF

	 25:
		 IF NOT arrAxisCtrl[AxiseNo.AxisName.SCurlingneedleWhirling].Io.biHomeSwitch  THEN
			  Mach_Control.WJ_b.Error[20]:=TRUE;//尾卷短卷针神伸缩回原点时,短卷针旋转原点传感器未亮报警
			  TailCurlStep1:=0;
		  ELSE 	 
			 TailCurlStep1:=30;
		 END_IF			
			

    30://尾卷长卷针伸缩轴回原点、尾卷短卷针伸缩轴回原点	
						IF NOT tTailCurlTON.Q THEN
								arrAxisCtrl[AxiseNo.AxisName.SCurlingneedleLine].Cmd.bHome:=TRUE;//尾卷短卷针平移回原点
								arrAxisCtrl[AxiseNo.AxisName.LCurlingneedleLine].Cmd.bHome:=TRUE;//尾卷长卷针平移回原点
								tTailCurlTON.IN:=TRUE;
						ELSE
								IF arrAxisCtrl[AxiseNo.AxisName.SCurlingneedleLine].Status.Homed AND arrAxisCtrl[AxiseNo.AxisName.SCurlingneedleLine].Status.NoMoving  AND
									 arrAxisCtrl[AxiseNo.AxisName.LCurlingneedleLine].Status.Homed AND arrAxisCtrl[AxiseNo.AxisName.LCurlingneedleLine].Status.NoMoving THEN
										arrAxisCtrl[AxiseNo.AxisName.SCurlingneedleLine].Cmd.bHome:=FALSE;//尾卷短卷针平移回原点
										arrAxisCtrl[AxiseNo.AxisName.LCurlingneedleLine].Cmd.bHome:=FALSE;//尾卷长卷针平移回原点
										tTailCurlTON.IN:=FALSE;
										TailCurlStep1:=35; 
								END_IF
						END_IF
			
		35:
						IF 	arrAxisCtrl[AxiseNo.AxisName.LCurlingneedleLine].Status.Homed AND arrAxisCtrl[AxiseNo.AxisName.LCurlingneedleLine].Status.NoMoving THEN
							IF arrAxisCtrl[AxiseNo.AxisName.LCurlingneedleLine].Cmd.arrbRealPoint[1] THEN
								arrAxisCtrl[AxiseNo.AxisName.LCurlingneedleLine].Cmd.iGoSetPos:=0;
							ELSE
								arrAxisCtrl[AxiseNo.AxisName.LCurlingneedleLine].Cmd.iGoSetPos:=1;//尾卷长卷针平移至初始位
							END_IF
						END_IF	
						IF 	arrAxisCtrl[AxiseNo.AxisName.SCurlingneedleLine].Status.Homed AND arrAxisCtrl[AxiseNo.AxisName.SCurlingneedleLine].Status.NoMoving THEN
							IF arrAxisCtrl[AxiseNo.AxisName.SCurlingneedleLine].Cmd.arrbRealPoint[1] THEN
								arrAxisCtrl[AxiseNo.AxisName.SCurlingneedleLine].Cmd.iGoSetPos:=0;
							ELSE
								arrAxisCtrl[AxiseNo.AxisName.SCurlingneedleLine].Cmd.iGoSetPos:=1;//尾卷短卷针平移至初始位
							END_IF
						END_IF		
							IF 	arrAxisCtrl[AxiseNo.AxisName.LCurlingneedleLine].Cmd.arrbRealPoint[1] AND arrAxisCtrl[AxiseNo.AxisName.LCurlingneedleLine].Status.NoMoving
								   AND arrAxisCtrl[AxiseNo.AxisName.SCurlingneedleLine].Cmd.arrbRealPoint[1] AND arrAxisCtrl[AxiseNo.AxisName.SCurlingneedleLine].Status.NoMoving THEN
									arrAxisCtrl[AxiseNo.AxisName.LCurlingneedleWhirling].Cmd.bHome:=FALSE;//尾卷长卷针旋转回原点
									arrAxisCtrl[AxiseNo.AxisName.SCurlingneedleWhirling].Cmd.bHome:=FALSE;//尾卷短卷针旋转回原点
									TailCurlStep1:=40; 
							END_IF
			
	40:
						IF 	arrAxisCtrl[AxiseNo.AxisName.LCurlingneedleLine].Cmd.arrbRealPoint[1] AND arrAxisCtrl[AxiseNo.AxisName.LCurlingneedleLine].Status.NoMoving AND
						arrAxisCtrl[AxiseNo.AxisName.LCurlingneedleLine].Cmd.arrbRealPoint[1] AND arrAxisCtrl[AxiseNo.AxisName.LCurlingneedleLine].Status.NoMoving THEN
						//IF NOT tTailCurlTON.Q THEN
								arrAxisCtrl[AxiseNo.AxisName.LCurlingneedleWhirling].Cmd.bHome:=TRUE;//尾卷长卷针旋转回原点
								arrAxisCtrl[AxiseNo.AxisName.SCurlingneedleWhirling].Cmd.bHome:=TRUE;//尾卷短卷针旋转回原点
								//tTailCurlTON.IN:=TRUE;
						//ELSE
								//IF arrAxisCtrl[AxiseNo.AxisName.LCurlingneedleWhirling].Status.Homed AND arrAxisCtrl[AxiseNo.AxisName.LCurlingneedleWhirling].Status.NoMoving AND 
								//	arrAxisCtrl[AxiseNo.AxisName.SCurlingneedleWhirling].Status.Homed AND arrAxisCtrl[AxiseNo.AxisName.SCurlingneedleWhirling].Status.NoMoving  THEN
									//tTailCurlTON.IN:=FALSE;
									TailCurlStep1:=50; 
								//END_IF	
						END_IF
	50://
					IF arrAxisCtrl[AxiseNo.AxisName.LCurlingneedleWhirling].Status.Homed AND arrAxisCtrl[AxiseNo.AxisName.LCurlingneedleWhirling].Status.NoMoving AND 
						arrAxisCtrl[AxiseNo.AxisName.SCurlingneedleWhirling].Status.Homed AND arrAxisCtrl[AxiseNo.AxisName.SCurlingneedleWhirling].Status.NoMoving  THEN
							TailCurlStep1:=51; 	
                            tTailCurlTON.IN:=FALSE;					
					END_IF
	51://夹电芯伸缩回原
			//IF arrAxisCtrl[AxiseNo.AxisName.TailCurlLine].Status.Homed AND arrAxisCtrl[AxiseNo.AxisName.TailCurlLine].Status.NoMoving THEN
				arrAxisCtrl[AxiseNo.AxisName.TailCurlRetracting].Cmd.bHome:=TRUE;//尾卷夹电芯伸缩回原点
				TailCurlStep1:=52; 
				tTailCurlTON.IN:=TRUE;
			//END_IF
	52:
		IF arrAxisCtrl[AxiseNo.AxisName.TailCurlRetracting].Status.Homed AND arrAxisCtrl[AxiseNo.AxisName.TailCurlRetracting].Status.NoMoving AND
           tTailCurlTON.Q  THEN
			arrAxisCtrl[AxiseNo.AxisName.TailCurlRetracting].Cmd.bHome:=FALSE;
			TailCurlStep1:=53; 
			tTailCurlTON.IN:=FALSE;
		END_IF					
					
	53://夹电芯平移回原
					IF 	arrAxisCtrl[AxiseNo.AxisName.LCurlingneedleLine].Cmd.arrbRealPoint[1] AND 	arrAxisCtrl[AxiseNo.AxisName.SCurlingneedleLine].Cmd.arrbRealPoint[1] AND 			
						arrAxisCtrl[AxiseNo.AxisName.SCurlingneedleLine].Status.Homed  AND   arrAxisCtrl[AxiseNo.AxisName.LCurlingneedleLine].Status.Homed  AND
						(arrAxisCtrl[AxiseNo.AxisName.TailCurlWhirling].Status.fSetPos<=arrAxisPar[AxiseNo.AxisName.TailCurlWhirling].arrTargetPoint[1]+1 AND
						arrAxisCtrl[AxiseNo.AxisName.TailCurlWhirling].Status.fSetPos>=arrAxisPar[AxiseNo.AxisName.TailCurlWhirling].arrTargetPoint[1]-1	) OR 
						(arrAxisCtrl[AxiseNo.AxisName.TailCurlWhirling].Status.fSetPos<=arrAxisPar[AxiseNo.AxisName.TailCurlWhirling].arrTargetPoint[2]+1 AND
						arrAxisCtrl[AxiseNo.AxisName.TailCurlWhirling].Status.fSetPos>=arrAxisPar[AxiseNo.AxisName.TailCurlWhirling].arrTargetPoint[2]-1	)  THEN
							arrAxisCtrl[AxiseNo.AxisName.TailCurlLine].Cmd.bHome:=TRUE;//尾卷夹电芯平移回原点
							TailCurlTorMark:=TRUE;//尾卷夹电芯平移力矩判断标志位
							TailCurlStep1:=54; 
							tTailCurlTON.IN:=TRUE;
                     ELSE
						    TailCurlStep1:=0; 
						     Mach_Control.WJ_b.Error[8]:=TRUE;//夹电芯平移回原点时条件不满足报警
					END_IF					
	54:
		IF arrAxisCtrl[AxiseNo.AxisName.TailCurlLine].Status.Homed AND arrAxisCtrl[AxiseNo.AxisName.TailCurlLine].Status.NoMoving AND
            tTailCurlTON.Q  THEN
			arrAxisCtrl[AxiseNo.AxisName.TailCurlLine].Cmd.bHome:=FALSE;
			TailCurlStep1:=60; 	
            tTailCurlTON.IN:=FALSE;	
		END_IF		
	
	60://夹电芯平移轴移至初始位、夹电芯伸缩轴移至初始位
						IF arrAxisCtrl[AxiseNo.AxisName.TailCurlLine].Status.Homed AND arrAxisCtrl[AxiseNo.AxisName.TailCurlLine].Status.NoMoving THEN
							TailCurlTorMark:=FALSE;//尾卷夹电芯平移力矩判断标志位
							IF arrAxisCtrl[AxiseNo.AxisName.TailCurlLine].Cmd.arrbRealPoint[1] THEN
								arrAxisCtrl[AxiseNo.AxisName.TailCurlLine].Cmd.iGoSetPos:=0;
							ELSE
								arrAxisCtrl[AxiseNo.AxisName.TailCurlLine].Cmd.iGoSetPos:=1;
							END_IF
						END_IF
						IF 	arrAxisCtrl[AxiseNo.AxisName.TailCurlRetracting].Status.Homed AND arrAxisCtrl[AxiseNo.AxisName.TailCurlRetracting].Status.NoMoving THEN
							IF arrAxisCtrl[AxiseNo.AxisName.TailCurlRetracting].Cmd.arrbRealPoint[1] THEN
								arrAxisCtrl[AxiseNo.AxisName.TailCurlRetracting].Cmd.iGoSetPos:=0;
							ELSE
								arrAxisCtrl[AxiseNo.AxisName.TailCurlRetracting].Cmd.iGoSetPos:=1;
							END_IF
						END_IF	
						IF arrAxisCtrl[AxiseNo.AxisName.TailCurlLine].Cmd.arrbRealPoint[1] AND  arrAxisCtrl[AxiseNo.AxisName.TailCurlLine].Status.NoMoving AND
							arrAxisCtrl[AxiseNo.AxisName.TailCurlRetracting].Cmd.arrbRealPoint[1] AND arrAxisCtrl[AxiseNo.AxisName.TailCurlRetracting].Status.NoMoving THEN
							TailCurlStep1:=70;
						END_IF
	70:		
			IF arrAxisCtrl[AxiseNo.AxisName.TailCurlLine].Cmd.arrbRealPoint[1] AND  arrAxisCtrl[AxiseNo.AxisName.TailCurlLine].Status.NoMoving AND
			arrAxisCtrl[AxiseNo.AxisName.TailCurlRetracting].Cmd.arrbRealPoint[1] AND arrAxisCtrl[AxiseNo.AxisName.TailCurlRetracting].Status.NoMoving THEN
			//IF NOT tTailCurlTON.Q THEN
				arrAxisCtrl[AxiseNo.AxisName.TailCurlUpDown].Cmd.bHome:=TRUE;//尾卷夹电芯升降回原点
				arrAxisCtrl[AxiseNo.AxisName.TailCurlSEPTAUpDown].Cmd.bHome:=TRUE;//尾卷夹膜升降回原点
				//tTailCurlTON.IN:=TRUE;
			//ELSE
				IF NOT  arrAxisCtrl[AxiseNo.AxisName.TailCurlUpDown].Status.Homed AND NOT arrAxisCtrl[AxiseNo.AxisName.TailCurlSEPTAUpDown].Status.Homed THEN
					TailCurlStep1:=75;
				END_IF
			END_IF	
	75:
		IF arrAxisCtrl[AxiseNo.AxisName.TailCurlUpDown].Status.Homed AND arrAxisCtrl[AxiseNo.AxisName.TailCurlUpDown].Status.NoMoving AND 
			arrAxisCtrl[AxiseNo.AxisName.TailCurlSEPTAUpDown].Status.Homed AND arrAxisCtrl[AxiseNo.AxisName.TailCurlSEPTAUpDown].Status.NoMoving THEN
			arrAxisCtrl[AxiseNo.AxisName.TailCurlUpDown].Cmd.bHome:=FALSE;//尾卷夹电芯升降回原点
			arrAxisCtrl[AxiseNo.AxisName.TailCurlSEPTAUpDown].Cmd.bHome:=FALSE;//尾卷夹膜升降回原点
			TailCurlStep1:=90;
		END_IF
    (*
    80:		
	     IF  arrAxisCtrl[AxiseNo.AxisName.TailCurlLine].Status.Homed AND arrAxisCtrl[AxiseNo.AxisName.TailCurlRetracting].Status.Homed AND
			 arrAxisCtrl[AxiseNo.AxisName.TailCurlLine].Cmd.arrbRealPoint[1] AND arrAxisCtrl[AxiseNo.AxisName.TailCurlRetracting].Cmd.arrbRealPoint[1] AND
             arrAxisCtrl[AxiseNo.AxisName.TailCurlWhirling].Status.fSetPos <5 (*AND NOT  arrAxisCtrl[AxiseNo.AxisName.TailCurlWhirling].Io.biHomeSwitch*) AND
             arrAxis[AxiseNo.AxisName.TailCurlWhirling].Status.Homed THEN
			      arrAxisPar[AxiseNo.AxisName.TailCurlWhirling].arrTargetPoint[10]:=5;
					IF arrAxisCtrl[AxiseNo.AxisName.TailCurlWhirling].Cmd.arrbRealPoint[10] AND NOT   arrAxis[AxiseNo.AxisName.TailCurlWhirling].Status.NotMoving THEN
						arrAxisCtrl[AxiseNo.AxisName.TailCurlWhirling].Cmd.iGoSetPos:=0;
						TailCurlWhirlTorMark:=FALSE;//尾卷夹电芯旋转力矩判断标志位
						TailCurlStep1:=81;
					ELSE
						arrAxisCtrl[AxiseNo.AxisName.TailCurlWhirling].Cmd.iGoSetPos:=10;
						TailCurlWhirlTorMark:=TRUE;//尾卷夹电芯旋转力矩判断标志位
					END_IF
		 END_IF
		 
	81:	
       IF arrAxis[AxiseNo.AxisName.TailCurlWhirling].Status.Homed  THEN
          arrAxisCtrl[AxiseNo.AxisName.TailCurlWhirling].Cmd.bHome:=TRUE;//尾卷夹旋转回原点
		  TailCurlWhirlTorMark:=TRUE;//尾卷夹电芯旋转力矩判断标志位
		  TailCurlStep1:=82;	
	 END_IF  
		
	82:	
      IF 	arrAxisCtrl[AxiseNo.AxisName.TailCurlWhirling].Status.Homed AND arrAxis[AxiseNo.AxisName.TailCurlWhirling].Status.NotMoving THEN	
		    arrAxisCtrl[AxiseNo.AxisName.TailCurlWhirling].Cmd.bHome:=FALSE;//尾卷夹旋转回原点
		    TailCurlStep1:=90;	
		   	TailCurlWhirlTorMark:=FALSE;//尾卷夹电芯旋转力矩判断标志位
	  END_IF
	 	IF   arrAxisCtrl[AxiseNo.AxisName.TailCurlWhirling].Status.fSetPos <-10 AND NOT arrAxisCtrl[AxiseNo.AxisName.TailCurlWhirling].Io.biHomeSwitch THEN
			 arrAxisCtrl[AxiseNo.AxisName.TailCurlWhirling].Cmd.bHome:=FALSE;//尾卷夹旋转回原点
			  arrAxisCtrl[AxiseNo.AxisName.TailCurlWhirling].Cmd.bStop:=TRUE;
			  TailCurlWhirlTorMark:=FALSE;//尾卷夹电芯旋转力矩判断标志位
			  TailCurlStep1:=9999;		
		END_IF		
		*)
 
	90://夹电芯旋转轴旋转至初始位
		IF 	arrAxis[AxiseNo.AxisName.TailCurlWhirling].Status.Homed AND arrAxis[AxiseNo.AxisName.TailCurlWhirling].Status.NotMoving AND
           arrAxisCtrl[AxiseNo.AxisName.TailCurlLine].Cmd.arrbRealPoint[1] AND arrAxisCtrl[AxiseNo.AxisName.TailCurlRetracting].Cmd.arrbRealPoint[1]  THEN
			IF arrAxisCtrl[AxiseNo.AxisName.TailCurlWhirling].Cmd.arrbRealPoint[1] THEN
				arrAxisCtrl[AxiseNo.AxisName.TailCurlWhirling].Cmd.iGoSetPos:=0;
				TailCurlWhirlTorMark:=FALSE;//尾卷夹电芯旋转力矩判断标志位
				TailCurlStep1:=100;
			ELSE
				arrAxisCtrl[AxiseNo.AxisName.TailCurlWhirling].Cmd.iGoSetPos:=1;
				TailCurlWhirlTorMark:=TRUE;//尾卷夹电芯旋转力矩判断标志位
			END_IF
		END_IF
	100://各轴移至初始位
		IF 	arrAxisCtrl[AxiseNo.AxisName.LCurlingneedleWhirling].Status.Homed AND arrAxisCtrl[AxiseNo.AxisName.LCurlingneedleWhirling].Status.NoMoving THEN
			IF arrAxisCtrl[AxiseNo.AxisName.LCurlingneedleWhirling].Cmd.arrbRealPoint[1] THEN
				arrAxisCtrl[AxiseNo.AxisName.LCurlingneedleWhirling].Cmd.iGoSetPos:=0;
			ELSE
				arrAxisCtrl[AxiseNo.AxisName.LCurlingneedleWhirling].Cmd.iGoSetPos:=1;//尾卷长卷针旋转至初始位
			END_IF
		END_IF				
		IF 	arrAxisCtrl[AxiseNo.AxisName.LCurlingneedleLine].Status.Homed AND arrAxisCtrl[AxiseNo.AxisName.LCurlingneedleLine].Status.NoMoving THEN
			IF arrAxisCtrl[AxiseNo.AxisName.LCurlingneedleLine].Cmd.arrbRealPoint[1] THEN
				arrAxisCtrl[AxiseNo.AxisName.LCurlingneedleLine].Cmd.iGoSetPos:=0;
			ELSE
				arrAxisCtrl[AxiseNo.AxisName.LCurlingneedleLine].Cmd.iGoSetPos:=1;//尾卷长卷针平移至初始位
			END_IF
		END_IF		
	
		IF 	arrAxisCtrl[AxiseNo.AxisName.SCurlingneedleWhirling].Status.Homed AND arrAxisCtrl[AxiseNo.AxisName.SCurlingneedleWhirling].Status.NoMoving THEN
			IF arrAxisCtrl[AxiseNo.AxisName.SCurlingneedleWhirling].Cmd.arrbRealPoint[1] THEN
				arrAxisCtrl[AxiseNo.AxisName.SCurlingneedleWhirling].Cmd.iGoSetPos:=0;
			ELSE
				arrAxisCtrl[AxiseNo.AxisName.SCurlingneedleWhirling].Cmd.iGoSetPos:=1;//尾卷短卷针旋转至初始位
			END_IF
		END_IF				
		IF 	arrAxisCtrl[AxiseNo.AxisName.SCurlingneedleLine].Status.Homed AND arrAxisCtrl[AxiseNo.AxisName.SCurlingneedleLine].Status.NoMoving THEN
			IF arrAxisCtrl[AxiseNo.AxisName.SCurlingneedleLine].Cmd.arrbRealPoint[1] THEN
				arrAxisCtrl[AxiseNo.AxisName.SCurlingneedleLine].Cmd.iGoSetPos:=0;
			ELSE
				arrAxisCtrl[AxiseNo.AxisName.SCurlingneedleLine].Cmd.iGoSetPos:=1;//尾卷短卷针平移至初始位
			END_IF
		END_IF		
				
		IF 	arrAxisCtrl[AxiseNo.AxisName.TailCurlSEPTAUpDown].Status.Homed AND arrAxisCtrl[AxiseNo.AxisName.TailCurlSEPTAUpDown].Status.NoMoving THEN
			IF arrAxisCtrl[AxiseNo.AxisName.TailCurlSEPTAUpDown].Cmd.arrbRealPoint[1] THEN
				arrAxisCtrl[AxiseNo.AxisName.TailCurlSEPTAUpDown].Cmd.iGoSetPos:=0;
			ELSE
				arrAxisCtrl[AxiseNo.AxisName.TailCurlSEPTAUpDown].Cmd.iGoSetPos:=1;//尾卷夹膜升降到初始位
			END_IF
		END_IF
		IF 	arrAxisCtrl[AxiseNo.AxisName.TailCurlUpDown].Status.Homed AND arrAxisCtrl[AxiseNo.AxisName.TailCurlUpDown].Status.NoMoving THEN
			IF arrAxisCtrl[AxiseNo.AxisName.TailCurlUpDown].Cmd.arrbRealPoint[1] THEN
				arrAxisCtrl[AxiseNo.AxisName.TailCurlUpDown].Cmd.iGoSetPos:=0;
			ELSE
				arrAxisCtrl[AxiseNo.AxisName.TailCurlUpDown].Cmd.iGoSetPos:=1;//尾卷夹电芯升降至初始位
			END_IF
		END_IF				
		IF arrAxisCtrl[AxiseNo.AxisName.LCurlingneedleWhirling].Cmd.arrbRealPoint[1] AND arrAxisCtrl[AxiseNo.AxisName.LCurlingneedleWhirling].Status.NoMoving AND 
			arrAxisCtrl[AxiseNo.AxisName.LCurlingneedleLine].Cmd.arrbRealPoint[1] AND arrAxisCtrl[AxiseNo.AxisName.LCurlingneedleLine].Status.NoMoving AND 
			arrAxisCtrl[AxiseNo.AxisName.LCurlingneedleWhirling].Cmd.arrbRealPoint[1] AND arrAxisCtrl[AxiseNo.AxisName.LCurlingneedleWhirling].Status.NoMoving AND 
			arrAxisCtrl[AxiseNo.AxisName.LCurlingneedleLine].Cmd.arrbRealPoint[1] AND arrAxisCtrl[AxiseNo.AxisName.LCurlingneedleLine].Status.NoMoving AND 
			arrAxisCtrl[AxiseNo.AxisName.TailCurlSEPTAUpDown].Cmd.arrbRealPoint[1] AND arrAxisCtrl[AxiseNo.AxisName.TailCurlSEPTAUpDown].Status.NoMoving AND 
			arrAxisCtrl[AxiseNo.AxisName.TailCurlUpDown].Cmd.arrbRealPoint[1] AND arrAxisCtrl[AxiseNo.AxisName.TailCurlUpDown].Status.NoMoving THEN
			TailCurlStep1:=110;
		END_IF	
	110://夹膜平移回初始位
				IF arrAxisCtrl[AxiseNo.AxisName.TailCurlSEPTALine].Cmd.arrbRealPoint[1] AND arrAxis[AxiseNo.AxisName.TailCurlSEPTALine].Status.NotMoving THEN	
							TailCurlStep1:=120;
							
				ELSE
							IF  arrAxisCtrl[AxiseNo.AxisName.TailCurlLine].Status.Homed AND arrAxisCtrl[AxiseNo.AxisName.TailCurlLine].Cmd.arrbRealPoint[1]
								AND arrAxisCtrl[AxiseNo.AxisName.CaDTCarryingUpDown].Cmd.arrbRealPoint[5]
                                (*TailCurlSEPTALineGoargee OR arrAxis[AxiseNo.AxisName.TailCurlSEPTALine].NcToPlc.SetPos<= arrAxisPar[AxiseNo.AxisName.TailCurlSEPTALine].arrTargetPoint[1]+50*) THEN	
									IF 	arrAxis[AxiseNo.AxisName.TailCurlSEPTALine].Status.Homed AND arrAxis[AxiseNo.AxisName.TailCurlSEPTALine].Status.NotMoving THEN
												IF arrAxisCtrl[AxiseNo.AxisName.TailCurlSEPTALine].Cmd.arrbRealPoint[1] THEN
													arrAxisCtrl[AxiseNo.AxisName.TailCurlSEPTALine].Cmd.iGoSetPos:=0;
													TailCurlSEPTATorMark:=FALSE;//夹膜平移力矩判断标志
												ELSE
													arrAxisCtrl[AxiseNo.AxisName.TailCurlSEPTALine].Cmd.iGoSetPos:=1;//尾卷夹膜平移至初始位
													TailCurlSEPTATorMark:=TRUE;//夹膜平移力矩判断标志
												END_IF
									END_IF		
							ELSE
										tTailCurlTON.IN:=FALSE;
										Mach_Control.WJ_b.Error[2]:=TRUE;//夹膜平移回原点条件不满足报警
										Tailcurl_Gohoming:=FALSE;//尾卷回原点中
										TailCurlStep1:=9999;		
							END_IF
				END_IF
				
	120://夹电芯平移去取电芯等待位		
			 IF arrAxisCtrl[AxiseNo.AxisName.TailCurlWhirling].Cmd.arrbRealPoint[1] AND arrAxisCtrl[AxiseNo.AxisName.TailCurlUpDown].Cmd.arrbRealPoint[1] AND
				arrAxisCtrl[AxiseNo.AxisName.TailCurlSEPTALine].Cmd.arrbRealPoint[1] AND  arrAxisCtrl[AxiseNo.AxisName.TailCurlSEPTAUpDown].Cmd.arrbRealPoint[1] AND
				arrAxisCtrl[AxiseNo.AxisName.LCurlingneedleLine].Cmd.arrbRealPoint[1] AND arrAxisCtrl[AxiseNo.AxisName.SCurlingneedleLine].Cmd.arrbRealPoint[1] AND
				arrCyCtrl[arrCyNo.CylinderName.PoleSplintCy_D].Io.DIOFFSwitch AND arrCyCtrl[arrCyNo.CylinderName.TailCurlUpdownCy].Io.DIOFFSwitch AND
				 arrAxisCtrl[AxiseNo.AxisName.TailCurlLine].Status.NoMoving   AND arrAxisCtrl[AxiseNo.AxisName.TailCurlWhirling].Cmd.arrbRealPoint[1]THEN
	 
					IF arrAxisCtrl[AxiseNo.AxisName.TailCurlLine].Cmd.arrbRealPoint[11]  THEN
						arrAxisCtrl[AxiseNo.AxisName.TailCurlLine].Cmd.iGoSetPos:=0;
						WZIniti_Done:=TRUE;//负极取片回原点完成
						Tailcurl_GohomeDone:=TRUE;//尾卷回原点完成
						Tailcurl_Gohoming:=FALSE;
						TailCurlStep1:=0;
						Mach_Control.WJ_b.TailCurlStep[1]:=0;
						TailCurlStep4:=0;
						TailCurlTorMark:=FALSE;//尾卷夹电芯平移力矩判断标志位
					ELSE
						arrAxisCtrl[AxiseNo.AxisName.TailCurlLine].Cmd.iGoSetPos:=11;//夹电芯平移移至取电芯等待位
						TailCurlTorMark:=TRUE;//尾卷夹电芯平移力矩判断标志位
					END_IF	
			 END_IF		
				
	END_CASE
	
END_IF

	IF Mach_Control.U.WJ_iMode=3 AND NOT arrAxisCtrl[AxiseNo.AxisName.TailCurlWhirling].Status.Homed AND arrAxis[AxiseNo.AxisName.TailCurlWhirling].Status.Moving AND
		arrAxisCtrl[AxiseNo.AxisName.TailCurlWhirling].Status.fSetPos <-10 AND TailCurlStep1<>82 AND  arrAxis[AxiseNo.AxisName.TailCurlWhirling].Status.Homed  THEN
	    arrAxisCtrl[AxiseNo.AxisName.TailCurlWhirling].Cmd.bHome:=FALSE;//尾卷夹旋转回原点
	    arrAxisCtrl[AxiseNo.AxisName.TailCurlWhirling].Cmd.bStop:=TRUE;
	END_IF
END_ACTION

ACTION TailCurlCam:
WJ_Cam_ton[1](PT:=T#100MS);
WJ_Cam_ton[2](PT:=T#100MS);
WJ_Cam_ton[3](PT:=T#100MS);
WJ_Cam_ton[4](PT:=T#100MS);
WJ_Cam_ton[5](PT:=T#100MS);

//尾卷凸轮曲线生成
CASE  iEndWindCam  OF   
10://计算相间距
    I20:=0;
    fMaxPosEndWind:=360;         // REAL
    fMinPosEndWind:=0;          //  REAL
    iNumberOfPointEndWind:=3600; //INT
    fIntervalEndWind:=(360-0)*0.5/ iNumberOfPointEndWind ;
    bEndWindCamDataEnable:=FALSE;
   	MEMSET(ADR(arrDeltaXmm),0,SIZEOF(arrDeltaXmm)); //  ARRAY[0..3600,0..1]  OF LREAL;  
    MEMSET(ADR(arrDeltaYmm),0,SIZEOF(arrDeltaYmm)); //  ARRAY[0..3600,0..1]  OF LREAL;  
    iEndWindCam:=20;  //INT

20:
   fbRoll_New.fAngleRel:=fAngleRel:=I20*fIntervalEndWind;
   bEndWindCamDataEnable:=TRUE;
    iEndWindCam:=30;

30:
   IF NOT  bEndWindCamDataEnable      THEN
           arrDeltaXmm[I20,0] := I20;
           arrDeltaXmm[I20,1] :=fbRoll_New.AxisXmm;

           arrDeltaYmm[I20,0] :=I20;
           arrDeltaYmm[I20,1] :=fbRoll_New.AxisYmm;

         I20:=I20+1;
		IF I20>iNumberOfPointEndWind THEN

			iEndWindCam:=666;  
		ELSE
               iEndWindCam:=20;  
		 END_IF
   END_IF

END_CASE


fbRoll_New(
	Enable:=bEndWindCamDataEnable , 
    fAngleRel:=fbRoll_New.fAngleRel,
	Width:= Par.Mechaical.fCellWidth , 
	Thick:=  Par.Mechaical.fCellThick, 
	r1:=        Par.Mechaical.fCellRadii  );
fbRoll_New.AxisXmm;
fbRoll_New.AxisYmm;



fbCreatCamEndWindX(
	Reset:=                               stSysState.bReset  , 
	bCreatTable:=                     fbCreatCamEndWindX.bCreatTable  , 
	iTable:=                             TableNo.M_TailCurlLine   , 
	arrCalculateTableData:=     arrDeltaXmm , 
	axisSlave:=                         arrAxis[AxiseNo.AxisName.TailCurlSEPTALine] , 
	axisMaster:=                      arrAxis[AxiseNo.VirAxisName.VirTailCurl] , 
	bCreatTableDone=> , 
	bCreatTableError=> , 
	bError=> );
  fbCreatCamEndWindX.bCreatTableDone;
  fbCreatCamEndWindX.bCreatTableError;
  fbCreatCamEndWindX.bError;


fbCreatCamEndWindY(
	Reset:=                               stSysState.bReset  , 
	bCreatTable:=                     fbCreatCamEndWindY.bCreatTable  , 
	iTable:=                            TableNo.M_TailCurlUpDown   , 
	arrCalculateTableData:=     arrDeltaYmm , 
	axisSlave:=                        arrAxis[AxiseNo.AxisName.TailCurlSEPTAUpDown] , 
	axisMaster:=                     arrAxis[AxiseNo.VirAxisName.VirTailCurl] , 
	bCreatTableDone=> , 
	bCreatTableError=> , 
	bError=> );
  fbCreatCamEndWindY.bCreatTableDone;
  fbCreatCamEndWindY.bCreatTableError;
  fbCreatCamEndWindY.bError;
  
 tWZCreateCamTON(IN:= , PT:=T#0.5S , Q=> , ET=> );
IF Mach_Control.U.DT_iMode=3 OR Mach_Control.U.DT_iMode=0 THEN//在手动状态下
				  //从触摸屏上创建尾卷凸轮
				  rWZCreateCam_TRIG(CLK:=Mach_Control.WJ_b.CreateCamStart , Q=> );
				  IF rWZCreateCam_TRIG.Q THEN
					  tWZCreateCamTON.IN:=FALSE;
					  WZCreatCamStep0:=10;
					  Mach_Control.WJ_b.Error[0]:=FALSE;
				  END_IF
END_IF				  
				  //尾卷凸轮创建自动程序
				  CASE WZCreatCamStep0 OF
							10:
									IF NOT   tWZCreateCamTON.Q THEN
											fbCreatCamEndWindX.bCreatTable :=FALSE;
											fbCreatCamEndWindY.bCreatTable:=FALSE;
											Mach_Control.WJ_b.CreateCamDone:=FALSE;
											tWZCreateCamTON.IN:=TRUE;
									ELSE
											tWZCreateCamTON.IN:=FALSE;
											WZCreatCamStep0:=11;
									END_IF
				  
							11:
									IF  NOT WJ_Cam_ton[1].Q THEN
										arrAxisCtrl[AxiseNo.AxisName.TailCurlSEPTALine].Cmd.bStop:=TRUE;
										arrAxisCtrl[AxiseNo.AxisName.TailCurlSEPTAUpDown].Cmd.bStop:=TRUE;
										WJ_Cam_ton[1].IN:=TRUE;
									ELSE
										WJ_Cam_ton[1].IN:=FALSE;
										WZCreatCamStep0:=12;
										arrAxisCtrl[AxiseNo.AxisName.TailCurlSEPTALine].Cmd.bStop:=FALSE;
										arrAxisCtrl[AxiseNo.AxisName.TailCurlSEPTAUpDown].Cmd.bStop:=FALSE;
									END_IF
					
							12:
									IF  NOT WJ_Cam_ton[2].Q THEN
										arrAxisCtrl[AxiseNo.AxisName.TailCurlSEPTALine].Cmd.bReset:=TRUE;	
										arrAxisCtrl[AxiseNo.AxisName.TailCurlSEPTAUpDown].Cmd.bReset:=TRUE;	
										WJ_Cam_ton[2].IN:=TRUE;
									 ELSE
										 WJ_Cam_ton[2].IN:=FALSE;
										 WZCreatCamStep0:=13;
										arrAxisCtrl[AxiseNo.AxisName.TailCurlSEPTALine].Cmd.bReset:=FALSE;	
										arrAxisCtrl[AxiseNo.AxisName.TailCurlSEPTAUpDown].Cmd.bReset:=FALSE;	
									 END_IF
									
							13:
									arrAxisCtrl[AxiseNo.AxisName.TailCurlSEPTALine].Cmd.bEnable:=TRUE;
									arrAxisCtrl[AxiseNo.AxisName.TailCurlSEPTAUpDown].Cmd.bEnable:=TRUE;
									IF arrAxisCtrl[AxiseNo.AxisName.TailCurlSEPTALine].Status.Enabled AND arrAxisCtrl[AxiseNo.AxisName.TailCurlSEPTAUpDown].Status.Enabled  THEN
										 WZCreatCamStep0:=20;
									END_IF		
						
				
									
							20://计算尾卷数据
									iEndWindCam:=10;
									Mach_Control.WJ_b.CreateCamDone:=FALSE;
									WZCreatCamStep0:=30;
							30://等持凸轮数据计算完成
								IF iEndWindCam=666 THEN
									WZCreatCamStep0:=40;
								END_IF
							40://创建尾卷平移凸轮，升降凸轮
									fbCreatCamEndWindX.bCreatTable :=TRUE;
									fbCreatCamEndWindY.bCreatTable:=TRUE;
									WZCreatCamStep0:=50;
							50://等待凸轮创建完成
									IF fbCreatCamEndWindX.bCreatTableDone AND fbCreatCamEndWindY.bCreatTableDone THEN
										Mach_Control.WJ_b.CreateCamDone:=TRUE;//尾卷凸轮创建完成
										WZCreatCamStep0:=6666;
									ELSE
											IF fbCreatCamEndWindX.bCreatTableError OR fbCreatCamEndWindY.bCreatTableError THEN
												Mach_Control.WJ_b.Error[0]:=TRUE;//尾卷凸轮创建失败
												WZCreatCamStep0:=6666;
											END_IF
									END_IF
				  END_CASE
(************************************************************凸轮耦合*****************************************************************************)
//夹膜平移凸轮耦合
//fbCamInEndWindX.ParCamIn.MasterScaling:=-0.05;
fbCamInEndWindX.ParCamIn.MasterScaling:=0.05;
fbCamInEndWindX.ParCamIn.SlaveScaling:=-1;
fbCamInEndWindX(  
	Reset:=                      stSysState.bReset  , 
	bCamInExecute:=       fbCamInEndWindX.bCamInExecute, 
	iTable1:=                   TableNo.M_TailCurlLine  , 
	ParCamIn:= , 
    axisMaster:=              arrAxis[AxiseNo.VirAxisName.VirTailCurl], 
	axisSlave:=                 arrAxis[AxiseNo.AxisName.TailCurlSEPTALine]   , 
	bError=> , 
	bReady=> , 
	bInSync=> );

P2M1_MachCtrl.WJ_b.Error[1]:=fbCamInEndWindX.bError;
fbCamInEndWindX.bReady;
fbCamInEndWindX.bInSync;
//夹膜升降凸轮耦合
fbCamInEndWindY.ParCamIn.MasterScaling:=0.05;
fbCamInEndWindY(  
	Reset:=                      stSysState.bReset  , 
	bCamInExecute:=       fbCamInEndWindY.bCamInExecute, 
	iTable1:=                   TableNo.M_TailCurlUpDown  , 
	ParCamIn:=               , 
    axisMaster:=              arrAxis[AxiseNo.VirAxisName.VirTailCurl], 
	axisSlave:=                arrAxis[AxiseNo.AxisName.TailCurlSEPTAUpDown]   , 
	bError=> , 
	bReady=> , 
	bInSync=> );

P2M1_MachCtrl.WJ_b.Error[2]:=fbCamInEndWindY.bError;
fbCamInEndWindY.bReady;
fbCamInEndWindY.bInSync;
(************************************************************齿轮耦合*****************************************************************************)
tailCurl1_GearIn(
	Master:=arrAxis[AxiseNo.VirAxisName.VirTailCurl] , 
	Slave:=arrAxis[AxiseNo.AxisName.SCurlingneedleWhirling] , 
	Execute:=tailCurl1_GearIn.Execute , 
	RatioNumerator:=1 , 
	RatioDenominator:=1 , 
	Acceleration:= , 
	Deceleration:= , 
	Jerk:= , 
	BufferMode:= , 
	Options:= , 
	InGear=> , 
	Busy=> , 
	Active=> , 
	CommandAborted=> , 
	Error=> , 
	ErrorID=> );
tailCurl1_GearIn.Error;
tailCurl1_GearIn.InGear;
	
	
fTailCurl2_TRIG(CLK:=tailCurl1_GearIn.Execute  , Q=> );
tailCurl2_CamOut(
	Slave:=arrAxis[AxiseNo.AxisName.SCurlingneedleWhirling], 
	Execute:=fTailCurl2_TRIG.Q , 
	Options:= , 
	Done=> , 
	Busy=> , 
	Error=> , 
	ErrorID=> );		
	
	
	
	
tailCurl2_GearIn(
	Master:=arrAxis[AxiseNo.VirAxisName.VirTailCurl]  , 
	Slave:=arrAxis[AxiseNo.AxisName.LCurlingneedleWhirling], 
	Execute:=tailCurl2_GearIn.Execute , 
	RatioNumerator:=1 , 
	RatioDenominator:=1 , 
	Acceleration:= , 
	Deceleration:= , 
	Jerk:= , 
	BufferMode:= , 
	Options:= , 
	InGear=> , 
	Busy=> , 
	Active=> , 
	CommandAborted=> , 
	Error=> , 
	ErrorID=> );
tailCurl2_GearIn.Error;
tailCurl2_GearIn.InGear;
	
fTailCurl3_TRIG(CLK:=tailCurl2_GearIn.Execute , Q=> );
tailCurl3_CamOut(
	Slave:=arrAxis[AxiseNo.AxisName.LCurlingneedleWhirling], 
	Execute:=fTailCurl3_TRIG.Q , 
	Options:= , 
	Done=> , 
	Busy=> , 
	Error=> , 
	ErrorID=> );
END_ACTION

ACTION TorqueCheckAlarm:
//力矩超限报警断使能
	IF 	Ca_Carrying1TorMark THEN//负极搬运1平移力矩判断标志位
		 IF arrAxisCtrl[AxiseNo.AxisName.CaCarryingLine1].Status.Moving AND (ABS(Torque.Ca_Carrying1Tor)>=Torque.Ca_Carrying1TorSet)  THEN
			Torque.Ca_Carrying1TorAlarm:=TRUE;
			arrAxisCtrl[AxiseNo.AxisName.CaCarryingLine1].Cmd.bEnable:=FALSE;
			//Ca_Carrying1TorMark:=FALSE;
			//Step_InitCaDT:=0;
		END_IF
	END_IF
	IF ABS(Torque.Ca_Carrying1Tor)<Torque.Ca_Carrying1TorSet AND Sys_Control.btn.System_Rrestbtn THEN
		Torque.Ca_Carrying1TorAlarm:=FALSE;
	END_IF
	
	IF 	Ca_Carrying2TorMark THEN//负极搬运2平移力矩判断标志位
		 IF arrAxisCtrl[AxiseNo.AxisName.CaCarryingLine2].Status.Moving AND (ABS(Torque.Ca_Carrying2Tor)>=Torque.Ca_Carrying2TorSet)  THEN
			Torque.Ca_Carrying2TorAlarm:=TRUE;
			arrAxisCtrl[AxiseNo.AxisName.CaCarryingLine2].Cmd.bEnable:=FALSE;
			//Ca_Carrying2TorMark:=FALSE;
			//Step_InitCaDT:=0;
		END_IF
	END_IF
	IF ABS(Torque.Ca_Carrying2Tor)<Torque.Ca_Carrying2TorSet AND Sys_Control.btn.System_Rrestbtn THEN
		Torque.Ca_Carrying2TorAlarm:=FALSE;
	END_IF
	
	IF 	Ca_DTCarryingTorMark THEN//负极叠台搬运平移力矩判断标志位	
		 IF arrAxisCtrl[AxiseNo.AxisName.CaDTCarryingLine].Status.Moving AND (ABS(Torque.Ca_DTCarryingTor)>=Torque.Ca_DTCarryingTorSet)  THEN
			Torque.Ca_DTCarryingTorAlarm:=TRUE;
			arrAxisCtrl[AxiseNo.AxisName.CaDTCarryingLine].Cmd.bEnable:=FALSE;
			//Ca_DTCarryingTorMark:=FALSE;
			//Step_InitCaDT:=0;
		END_IF
	END_IF
	IF ABS(Torque.Ca_DTCarryingTor)<Torque.Ca_DTCarryingTorSet AND Sys_Control.btn.System_Rrestbtn THEN
		Torque.Ca_DTCarryingTorAlarm:=FALSE;
	END_IF	

//力矩超限报警断使能
	IF 	An_CarryingTorMark THEN//正极搬运1移位力矩判断标志位
		 IF arrAxisCtrl[AxiseNo.AxisName.AnCarryingLine].Status.Moving AND (ABS(Torque.An_CarryingTor)>=Torque.An_CarryingTorSet)  THEN
			Torque.An_CarryingTorAlarm:=TRUE;
			arrAxisCtrl[AxiseNo.AxisName.AnCarryingLine].Cmd.bEnable:=FALSE;
			//An_CarryingTorMark:=FALSE;//正极搬运1移位力矩判断标志位
			//Step_InitAnDT:=0;
		END_IF
	END_IF
	IF ABS(Torque.An_CarryingTor)<Torque.An_CarryingTorSet AND Sys_Control.btn.System_Rrestbtn THEN
		Torque.An_CarryingTorAlarm:=FALSE;
	END_IF
	
	IF 	An_DTCarryingTorMark THEN//正极叠台搬运力矩判断标志位	
		 IF arrAxisCtrl[AxiseNo.AxisName.AnDTCarryingLine].Status.Moving AND (ABS(Torque.An_DTCarryingTor)>=Torque.Ca_Carrying1TorSet)  THEN
			Torque.An_DTCarryingTorAlarm:=TRUE;
			arrAxisCtrl[AxiseNo.AxisName.AnDTCarryingLine].Cmd.bEnable:=FALSE;
			An_DTCarryingTorMark:=FALSE;//正极叠台搬运力矩判断标志位	
			//Step_InitAnDT:=0;
		END_IF
	END_IF
	IF ABS(Torque.An_DTCarryingTor)<Torque.Ca_Carrying1TorSet AND Sys_Control.btn.System_Rrestbtn THEN
		Torque.An_DTCarryingTorAlarm:=FALSE;
	END_IF
	
//力矩超限报警断使能
	IF 	TailCurlTorMark THEN//尾卷夹电芯平移力矩判断标志位
		 IF arrAxisCtrl[AxiseNo.AxisName.TailCurlLine].Status.Moving AND (ABS(Torque.TailCurlTor)>=Torque.TailCurlTorSet)  THEN
			Torque.TailCurlTorAlarm:=TRUE;
			arrAxisCtrl[AxiseNo.AxisName.TailCurlLine].Cmd.bEnable:=FALSE;
			//TailCurlTorMark:=FALSE;
			//TailCurlStep1:=0;
		END_IF
	END_IF
	IF ABS(Torque.TailCurlTor)<Torque.TailCurlTorSet AND Sys_Control.btn.System_Rrestbtn THEN
		Torque.TailCurlTorAlarm:=FALSE;
	END_IF
	
	IF 	TailCurlWhirlTorMark THEN//尾卷夹电芯旋转力矩判断标志位
		 IF arrAxisCtrl[AxiseNo.AxisName.TailCurlWhirling].Status.Moving AND (ABS(Torque.TailCurlWhirlTor)>=Torque.TailCurlWhirlTorSet)  THEN
			Torque.TailCurlWhirlTorAlarm:=TRUE;
			arrAxisCtrl[AxiseNo.AxisName.TailCurlWhirling].Cmd.bEnable:=FALSE;
			//TailCurlWhirlTorMark:=FALSE;
			//TailCurlStep1:=0;
		END_IF
	END_IF
	IF ABS(Torque.TailCurlWhirlTor)<Torque.TailCurlWhirlTorSet AND Sys_Control.btn.System_Rrestbtn THEN
		Torque.TailCurlWhirlTorAlarm:=FALSE;
	END_IF

	IF 	TailCurlSEPTATorMark THEN//夹膜平移力矩判断标志位
		 IF arrAxisCtrl[AxiseNo.AxisName.TailCurlSEPTALine].Status.Moving AND (ABS(Torque.TailCurlSEPTATor)>=Torque.TailCurlSEPTATorSet)  THEN
			Torque.TailCurlSEPTATorAlarm:=TRUE;
			arrAxisCtrl[AxiseNo.AxisName.TailCurlSEPTALine].Cmd.bEnable:=FALSE;
			//TailCurlSEPTATorMark:=FALSE;
			//TailCurlStep1:=0;
		END_IF
	END_IF
	IF ABS(Torque.TailCurlSEPTATor)<Torque.TailCurlSEPTATorSet AND Sys_Control.btn.System_Rrestbtn THEN
		Torque.TailCurlSEPTATorAlarm:=FALSE;
	END_IF	
(*
	IF 	TailCurlRetMark THEN//尾卷夹电芯伸缩力矩判断标志	
		 IF arrAxisCtrl[AxiseNo.AxisName.TailCurlRetracting].Status.Moving AND (ABS(Torque.TailCurlRetTor)>=Torque.TailCurlRetTorSet)  THEN
			Torque.TailCurlRetTorAlarm:=TRUE;
			arrAxisCtrl[AxiseNo.AxisName.TailCurlRetracting].Cmd.bEnable:=FALSE;
			//TailCurlRetMark:=FALSE;
			//TailCurlStep1:=0;
		END_IF
	END_IF
	IF ABS(Torque.TailCurlRetTor)<Torque.TailCurlRetTorSet AND Sys_Control.btn.System_Rrestbtn THEN
		Torque.TailCurlRetTorAlarm:=FALSE;
	END_IF	
*)
END_ACTION

ACTION Vacuum_Signal:
(**************************************************分段皮带***********************************************************)
(*
//正极模切送料分段皮带
fbAnBeltVacuum( Vacuumsel:= , 
						   	tPTtime:= , 	
							VarrCyCtrl1:=arrCyCtrl[arrCyNo.ElectValveName.AnBeltVacuum] , 
							VarrCyCtrl2:=arrCyCtrl[arrCyNo.ElectValveName.AnBeltVacuumBark] );

//负极模切送料分段皮带
fbCaMQBeltVacuum(Vacuumsel:= , 
								tPTtime:= , 
								VarrCyCtrl1:=arrCyCtrl[arrCyNo.ElectValveName.CaMQBeltVacuum] , 
								VarrCyCtrl2:=arrCyCtrl[arrCyNo.ElectValveName.CaMQBeltVacuumBark] );

//负极送片皮带末端真空
fbCaLoadUpBeltVacuum(Vacuumsel:= , 
										tPTtime:= , 
										VarrCyCtrl1:=arrCyCtrl[arrCyNo.ElectValveName.CaLoadUpBeltVacuum] , 
										VarrCyCtrl2:=arrCyCtrl[arrCyNo.ElectValveName.CaLoadUpBeltVacuumBark] );




(**************************************************叠片吸盘***********************************************************)
//正极送片搬运升降真空
fbAnCarryingVacuum(Vacuumsel:= , 
									tPTtime:= , 
									VarrCyCtrl1:=arrCyCtrl[arrCyNo.ElectValveName.AnCarryingVacuum] , 
									VarrCyCtrl2:=arrCyCtrl[arrCyNo.ElectValveName.AnCarryingVacuumBark] );

//正极叠片搬运升降真空
fbAnDTCarryingVacuum(Vacuumsel:= , 
										tPTtime:= , 
										VarrCyCtrl1:=arrCyCtrl[arrCyNo.ElectValveName.AnDTCarryingVacuum] , 
										VarrCyCtrl2:=arrCyCtrl[arrCyNo.ElectValveName.AnDTCarryingVacuumBark] );

//正极纠偏平台真空
fbAndeviationVacuum(Vacuumsel:= , 
									tPTtime:= , 
									VarrCyCtrl1:=arrCyCtrl[arrCyNo.ElectValveName.AndeviationVacuum] , 
									VarrCyCtrl2:=arrCyCtrl[arrCyNo.ElectValveName.AndeviationVacuumBark] );

									
//负极送片搬运升降1真空
fbCaCarryingVacuum1(Vacuumsel:= , 
									tPTtime:= , 
									VarrCyCtrl1:=arrCyCtrl[arrCyNo.ElectValveName.CaCarryingVacuum1], 
									VarrCyCtrl2:=arrCyCtrl[arrCyNo.ElectValveName.CaCarryingVacuumBark1] );

//负极送片搬运升降2真空
fbCaCarryingVacuum2(Vacuumsel:= , 
									tPTtime:= , 
									VarrCyCtrl1:=arrCyCtrl[arrCyNo.ElectValveName.CaCarryingVacuum2] , 
									VarrCyCtrl2:=arrCyCtrl[arrCyNo.ElectValveName.CaCarryingVacuumBark2] );
 
//负极叠片搬运升降真空
fbCaDTCarryingVacuum(Vacuumsel:= , 
										tPTtime:= , 
										VarrCyCtrl1:=arrCyCtrl[arrCyNo.ElectValveName.CaDTCarryingVacuum] , 
										VarrCyCtrl2:=arrCyCtrl[arrCyNo.ElectValveName.CaDTCarryingVacuumBark] );
 
//负极纠偏平台真空
fbCadeviationVacuum(Vacuumsel:= , 
									tPTtime:= , 
									VarrCyCtrl1:=arrCyCtrl[arrCyNo.ElectValveName.CadeviationVacuum] , 
									VarrCyCtrl2:=arrCyCtrl[arrCyNo.ElectValveName.CadeviationVacuumBark] );

*)


(***********************************正极分段皮带皮带末端真空控制*******************************************)
(*
//正极取料中,模切皮带破真空V1
IF Mach_Control.An_b.An_MainBelting THEN
	IF arrAxisCtrl[AxiseNo.AxisName.AnCarryingUpDown].Cmd.arrbRealPoint[2] THEN
		//fbAnBeltVacuum.Vacuumsel:=2;//正极模切送料分段皮带破真空开
		arrCyCtrl[arrCyNo.ElectValveName.AnBeltVacuumBark].Cmd.bON:=TRUE;//正极模切送料分段皮带破真空打开
		arrCyCtrl[arrCyNo.ElectValveName.AnBeltVacuumBark].Cmd.bOFF:=FALSE;//正极模切送料分段皮带破真空打关
	END_IF
ELSIF Mach_Control.An_b.AN_BeltDone OR Mach_Control.U.Step[0]=20 THEN //OR Mach_Control.U.DT_iMode = 1 
	arrCyCtrl[arrCyNo.ElectValveName.AnBeltVacuumBark].Cmd.bON:=FALSE;//正极模切送料分段皮带破真空打开
	arrCyCtrl[arrCyNo.ElectValveName.AnBeltVacuumBark].Cmd.bOFF:=TRUE;//正极模切送料分段皮带破真空打关
	//fbAnBeltVacuum.Vacuumsel:=1;//正极模切送料分段皮带真空打开	
END_IF	
*)	

///V2
rtVacuum2(CLK:=Mach_Control.An_b.An_MainBelting  , Q=> );
ftVacuum2(CLK:=Mach_Control.An_b.An_MainBelting    , Q=> );
IF  rtVacuum2.Q THEN//破真空
      arrCyCtrl[arrCyNo.ElectValveName.AnBeltVacuumBark].Cmd.bON:=TRUE;//正极模切送料分段皮带破真空打开
     arrCyCtrl[arrCyNo.ElectValveName.AnBeltVacuumBark].Cmd.bOFF:=FALSE;//正极模切送料分段皮带破真空打关
END_IF
IF  ftVacuum2.Q THEN//开真空
     arrCyCtrl[arrCyNo.ElectValveName.AnBeltVacuumBark].Cmd.bOFF:=TRUE;//正极模切送料分段皮带破真空打关
    arrCyCtrl[arrCyNo.ElectValveName.AnBeltVacuumBark].Cmd.bON:=FALSE;//正极模切送料分段皮带破真空打开
END_IF




(***********************************负极分段皮带皮带末端真空控制*******************************************)
(*
//负极取料中,模切皮带破真空V1
IF Mach_Control.Ca_b.Ca_MainBelting THEN
	IF arrAxisCtrl[AxiseNo.AxisName.CaCarryingUpDown1].Cmd.arrbRealPoint[1] THEN
		arrCyCtrl[arrCyNo.ElectValveName.CaMQBeltVacuumBark].Cmd.bON:=TRUE;//负极送片皮带末端真空开	
		arrCyCtrl[arrCyNo.ElectValveName.CaMQBeltVacuumBark].Cmd.bOFF:=FALSE;//负极送片皮带末端真空关	
		//fbCaMQBeltVacuum.Vacuumsel:=2;//负极模切分段皮带破真空开
	END_IF	
ELSIF Mach_Control.Ca_b.Ca_BeltDone  OR Mach_Control.U.Step[0]=20 THEN //OR Mach_Control.U.DT_iMode = 1
	arrCyCtrl[arrCyNo.ElectValveName.CaMQBeltVacuumBark].Cmd.bON:=FALSE;//负极送片皮带末端真空开	
	arrCyCtrl[arrCyNo.ElectValveName.CaMQBeltVacuumBark].Cmd.bOFF:=TRUE;//负极送片皮带末端真空关	
	//fbCaMQBeltVacuum.Vacuumsel:=1;//负极模切分段皮带真空打开
END_IF
*)

///V2
rtVacuum3(CLK:=Mach_Control.Ca_b.Ca_MainBelting  , Q=> );
ftVacuum3(CLK:=Mach_Control.Ca_b.Ca_MainBelting    , Q=> );
IF  rtVacuum3.Q THEN//破真空
		arrCyCtrl[arrCyNo.ElectValveName.CaMQBeltVacuumBark].Cmd.bON:=TRUE;//负极模切分段皮带破真空打开
		arrCyCtrl[arrCyNo.ElectValveName.CaMQBeltVacuumBark].Cmd.bOFF:=FALSE;//负极模切分段皮带破真空打关
END_IF
IF  ftVacuum3.Q THEN//开真空
		arrCyCtrl[arrCyNo.ElectValveName.CaMQBeltVacuumBark].Cmd.bOFF:=TRUE;//负极模切分段皮带破真空打关
		arrCyCtrl[arrCyNo.ElectValveName.CaMQBeltVacuumBark].Cmd.bON:=FALSE;//负极模切分段皮带破真空打开
END_IF



(*******************************************负极缓存皮带末端真空控制**************************************************)
//负极送片搬运输出取片中 打开破真空      取片搬运复位开真空此时吸盘离开皮带5mm          
(*
//负极取料中,缓存皮带破真空V1
IF NOT  Mach_Control.U.EmptyRunMode  THEN
	IF Mach_Control.Ca_b.Ca_CacheBelting THEN
		
		IF arrAxisCtrl[AxiseNo.AxisName.CaCarryingUpDown2].Cmd.arrbRealPoint[2] THEN
			arrCyCtrl[arrCyNo.ElectValveName.CaLoadUpBeltVacuumBark].Cmd.bON:=TRUE;//负极送片皮带末端真空开	
			arrCyCtrl[arrCyNo.ElectValveName.CaLoadUpBeltVacuumBark].Cmd.bOFF:=FALSE;//负极送片皮带末端真空关	
			//fbCaLoadUpBeltVacuum.Vacuumsel:=2;//负极送片皮带末端破真空开
		END_IF
	ELSIF arrAxisCtrl[AxiseNo.AxisName.CaBelt].Status.Moving  OR Mach_Control.U.Step[0]=20 THEN //OR Mach_Control.U.DT_iMode = 1
		arrCyCtrl[arrCyNo.ElectValveName.CaLoadUpBeltVacuumBark].Cmd.bON:=FALSE;//负极送片皮带末端真空开	
		arrCyCtrl[arrCyNo.ElectValveName.CaLoadUpBeltVacuumBark].Cmd.bOFF:=TRUE;//负极送片皮带末端真空关	
		//fbCaLoadUpBeltVacuum.Vacuumsel:=1;//负极送片皮带末端真空开
	END_IF
END_IF
*)

arrCyCtrl[arrCyNo.ElectValveName.CaLoadUpBeltVacuumBark].Status.OFFState;
arrCyCtrl[arrCyNo.ElectValveName.CaLoadUpBeltVacuumBark].Status.ONState;
///V2
rtVacuum1(CLK:=Mach_Control.Ca_b.Ca_CacheBelting , Q=> );
ftVacuum1(CLK:=Mach_Control.Ca_b.Ca_CacheBelting , Q=> );
	IF rtVacuum1.Q THEN
		arrCyCtrl[arrCyNo.ElectValveName.CaLoadUpBeltVacuumBark].Cmd.bOFF:=FALSE;//负极送片皮带末端真空关
		arrCyCtrl[arrCyNo.ElectValveName.CaLoadUpBeltVacuumBark].Cmd.bON:=TRUE;//负极送片皮带末端真空开
	END_IF
	IF ftVacuum1.Q THEN
		arrCyCtrl[arrCyNo.ElectValveName.CaLoadUpBeltVacuumBark].Cmd.bOFF:=TRUE;//负极送片皮带末端真空关
		arrCyCtrl[arrCyNo.ElectValveName.CaLoadUpBeltVacuumBark].Cmd.bON:=FALSE;//负极送片皮带末端真空开
	END_IF











  //  arrAxisCtrl[AxiseNo.AxisName.CaCarryingUpDown2].Status.fActPos<= arrAxisPar[AxiseNo.AxisName.CaCarryingUpDown2].arrTargetPoint[2]-5



(*
IF  Mach_Control.U.EmptyRunMode  THEN
	IF Mach_Control.Ca_b.Ca_CacheBelting AND  arrAxisCtrl[AxiseNo.AxisName.CaCarryingUpDown2].Cmd.arrbRealPoint[2] AND
		NOT arrAxisCtrl[AxiseNo.AxisName.CaBelt].Status.Moving THEN
		arrCyCtrl[arrCyNo.ElectValveName.CaLoadUpBeltVacuumBark].Cmd.bON:=TRUE;//负极送片皮带末端真空开	
		arrCyCtrl[arrCyNo.ElectValveName.CaLoadUpBeltVacuumBark].Cmd.bOFF:=FALSE;//负极送片皮带末端真空关	
		//fbCaLoadUpBeltVacuum.Vacuumsel:=2;//负极送片皮带末端破真空开
	ELSIF arrAxisCtrl[AxiseNo.AxisName.CaBelt].Status.Moving  OR Mach_Control.U.Step[0]=20 THEN
		arrCyCtrl[arrCyNo.ElectValveName.CaLoadUpBeltVacuumBark].Cmd.bON:=FALSE;//负极送片皮带末端真空开	
		arrCyCtrl[arrCyNo.ElectValveName.CaLoadUpBeltVacuumBark].Cmd.bOFF:=TRUE;//负极送片皮带末端真空关	
		//fbCaLoadUpBeltVacuum.Vacuumsel:=1;//负极送片皮带末端真空开
	END_IF
END_IF	
*)
	

(*
//正极取料中,模切皮带破真空
IF Mach_Control.An_b.An_MainBelting THEN
	IF arrAxisCtrl[AxiseNo.AxisName.AnCarryingUpDown].Cmd.arrbRealPoint[2] THEN
		fbAnBeltVacuum.Vacuumsel:=2;//正极模切送料分段皮带破真空开
	END_IF
ELSIF Mach_Control.An_b.AN_BeltDone OR Mach_Control.U.DT_iMode = 1 OR Mach_Control.U.Step[0]=20 THEN
	fbAnBeltVacuum.Vacuumsel:=1;//正极模切送料分段皮带真空打开	
END_IF		

//负极取料中,模切皮带破真空
IF Mach_Control.Ca_b.Ca_MainBelting THEN
	IF arrAxisCtrl[AxiseNo.AxisName.CaCarryingUpDown1].Cmd.arrbRealPoint[1] THEN
		fbCaMQBeltVacuum.Vacuumsel:=2;//负极模切分段皮带破真空开
	END_IF	
ELSIF Mach_Control.Ca_b.Ca_BeltDone OR Mach_Control.U.DT_iMode = 1 OR Mach_Control.U.Step[0]=20 THEN
	fbCaMQBeltVacuum.Vacuumsel:=1;//负极模切分段皮带真空打开
END_IF


	//正极取料中,控制皮带破真空
	IF Mach_Control.An_b.An_MainBelting   THEN//AND Mach_Control.An_b.An_MainBeltOK 
			arrCyCtrl[arrCyNo.ElectValveName.AnBeltVacuumBark].Cmd.bON:=TRUE;//正极模切送料分段皮带破真空打开
			arrCyCtrl[arrCyNo.ElectValveName.AnBeltVacuumBark].Cmd.bOFF:=FALSE;//正极模切送料分段皮带破真空打关
	ELSE
			arrCyCtrl[arrCyNo.ElectValveName.AnBeltVacuumBark].Cmd.bOFF:=TRUE;//正极模切送料分段皮带破真空打关
			arrCyCtrl[arrCyNo.ElectValveName.AnBeltVacuumBark].Cmd.bON:=FALSE;//正极模切送料分段皮带破真空打开
	END_IF
	//负极取料中,控制皮带破真空
	IF Mach_Control.Ca_b.Ca_MainBelting   THEN//AND Mach_Control.Ca_b.Ca_MainBeltOK 
		arrCyCtrl[arrCyNo.ElectValveName.CaMQBeltVacuumBark].Cmd.bON:=TRUE;//负极模切分段皮带破真空打开
		arrCyCtrl[arrCyNo.ElectValveName.CaMQBeltVacuumBark].Cmd.bOFF:=FALSE;//负极模切分段皮带破真空打关
	ELSE
		arrCyCtrl[arrCyNo.ElectValveName.CaMQBeltVacuumBark].Cmd.bOFF:=TRUE;//负极模切分段皮带破真空打关
		arrCyCtrl[arrCyNo.ElectValveName.CaMQBeltVacuumBark].Cmd.bON:=FALSE;//负极模切分段皮带破真空打开
	END_IF
	IF(* Mach_Control.Ca_b.Ca_CacheBelting  AND *)Mach_Control.Ca_b.Ca_CacheBeltDLOK AND arrAxisCtrl[AxiseNo.AxisName.CaBelt].Status.NoMoving THEN
		arrCyCtrl[arrCyNo.ElectValveName.CaLoadUpBeltVacuumBark].Cmd.bOFF:=FALSE;//负极送片皮带末端真空关
		arrCyCtrl[arrCyNo.ElectValveName.CaLoadUpBeltVacuumBark].Cmd.bON:=TRUE;//负极送片皮带末端真空开					
	ELSE
		arrCyCtrl[arrCyNo.ElectValveName.CaLoadUpBeltVacuumBark].Cmd.bOFF:=TRUE;//负极送片皮带末端真空关
		arrCyCtrl[arrCyNo.ElectValveName.CaLoadUpBeltVacuumBark].Cmd.bON:=FALSE;//负极送片皮带末端真空开
	END_IF
*)
END_ACTION

ACTION WJ_SingMode:
						IF Mach_Control.TJ_b.SinStepMode THEN//尾卷单步模式
							TailCurlSinStep:=TRUE;
						ELSE
							TailCurlSinStep:=FALSE;
						END_IF
END_ACTION

END_FUNCTION_BLOCK

// ---- P2POUs/BasicFunction/05_Actuators/FB_Vacuum.TcPOU
FUNCTION_BLOCK FB_Vacuum
VAR_INPUT
	Vacuumsel:BYTE:=0;//0=真空和破真空都关，1=真空开，2=破真空开。
	tPTtime:TIME:=T#600MS;
END_VAR

VAR_IN_OUT
	VarrCyCtrl1			                  :ST_CyCtrl;//真空
	VarrCyCtrl2			                  :ST_CyCtrl;//破真空		
END_VAR

VAR
	ton:TON;	
END_VAR

ton(IN:= , PT:=tPTtime , Q=> , ET=> );
IF Vacuumsel=0  THEN
	VarrCyCtrl1.Cmd.bON:=VarrCyCtrl2.Cmd.bON:=FALSE;
	VarrCyCtrl1.Cmd.bOFF:=VarrCyCtrl2.Cmd.bOFF:=TRUE;
	ton.IN:=FALSE;
	Vacuumsel:=3;
ELSIF Vacuumsel=1 THEN
	VarrCyCtrl1.Cmd.bON:=VarrCyCtrl2.Cmd.bOFF:=TRUE;
	VarrCyCtrl1.Cmd.bOFF:=VarrCyCtrl2.Cmd.bON:=FALSE;
	ton.IN:=FALSE;
	Vacuumsel:=3;	
ELSIF Vacuumsel=2  THEN
	VarrCyCtrl1.Cmd.bON:=VarrCyCtrl2.Cmd.bOFF:=FALSE;
	VarrCyCtrl1.Cmd.bOFF:=VarrCyCtrl2.Cmd.bON:=TRUE;
	ton.IN:=TRUE;
	IF ton.Q THEN
		ton.IN:=FALSE;
		Vacuumsel:=0;
	END_IF	
END_IF

END_FUNCTION_BLOCK

// ---- P2POUs/BasicFunction/12_User2/Rectifydev_PID.TcPOU
FUNCTION_BLOCK Rectifydev_PID
VAR_INPUT
	Enable:BOOL;//启动条件
	RestHMI:BOOL;//报警复位
	MasterNo:UINT;//主轴号
	SlaveNo1:UINT;//从轴号1
	SlaveNo2:UINT;//从轴号2
	MasterValue:REAL;//主轴匀速运行时的速度
	RecDevagree:BOOL;//纠偏许可
	RecDevEqupos:REAL;//纠偏平传感器的平衡位置
	RecDevValueSet:REAL;//纠偏偏差量设定
	RecDevPV:REAL;//纠偏传感器当前值
	RecDevSpeedCoe:REAL;//纠偏带速度系数
	CWW:BOOL;//纠偏方向选择
	AxisPos_H:REAL;//从轴的纠偏行程上限
	AxisPos_L:REAL;//从轴的纠偏行程下限
END_VAR
VAR_OUTPUT
	RecDevSpeed:REAL;//纠偏速度
	Error:ARRAY[0..9] OF BOOL;//报警
END_VAR
VAR
	// 执行延时2S
	TON1: TON;
	// 轴纠偏上限
	AxisRecDevPos_H: REAL;
	// 轴的纠偏下限
	AxisRecDevPos_L: REAL;
	// 从轴1的当前位置
	AxisRecDevActPos1: LREAL;
	// 从轴2的当前位置
	AxisRecDevActPos2: LREAL;
	// 从轴1纠偏超限
	PosOverLimit1: BOOL;
	// 从轴2纠偏超限
	PosOverLimit2: BOOL;
	
	// 纠偏传感器上限值
	RecDevSensors_H: REAL;
	// 纠偏传感器下限值
	RecDevSensors_L: REAL;
	// 纠偏轴的速度
	MC_RecDevvelocity: REAL;
	// 纠偏轴的中间速度
	MC_RecDevvelocity_M: REAL;
	// 轴纠偏允许
	MC_RecDevagree: BOOL;
	RecDev_GearInDyn: MC_GearInDyn;
	// 主轴解除耦合

	// 主轴停止
	Master_Stop: MC_Stop;
	// 从轴解除耦合
	SlaveCamOut: MC_CamOut;
	// 主轴匀速运动
	MasterMoveVelocity: MC_MoveVelocity;
	sR_TRIG: R_TRIG;
	sF_TRIG: F_TRIG;
	Slave_Stop: MC_Stop;
	Step0: INT;
	// 主、从轴停止
	AxisStop: BOOL;
	GearInMultiMaster: MC_GearInMultiMaster;
	TON2: TON;
	GearInMultiMaster1: MC_GearInMultiMaster;
	SlaveCamOut2: MC_CamOut;
	Slave_Stop2: MC_STOP;
END_VAR

TON1(IN:=Enable , PT:=T#2S , Q=> , ET=> );//执行延时2S
TON2(IN:=Enable , PT:=T#10S , Q=> , ET=> );//纠偏凸轮耦合超时
sR_TRIG(CLK:=Enable , Q=> );
sF_TRIG(CLK:=Enable , Q=> );

(**************************纠偏传感器的纠偏范围,大于最大值，小于最小值开始纠偏 *****************************)
RecDevSensors_H:=RecDevEqupos+RecDevValueSet;//纠偏传感器上限值(如果，纠偏传感器的当前值在上、下限这冗余，就不纠一万)
RecDevSensors_L:=RecDevEqupos-RecDevValueSet;//纠偏传感器下限值

